    if(wv_seq[0] == 0 or wv_seq[0] == 3):
      if(a9_wv_weldingon==True):
        program_weld_on = False
        if(isHicomm):
          write_port_register(202,0)
          write_port_register(149,0)
        else:
          set_standard_digital_out(0,False)
        end
        if(wv_weldpar[2]==1):
          target_pos = feature_offset(get_actual_tcp_pose(),p[0,0,-0.01,0,0,0],wv_Line_Feature2)
          movel(target_pos,0.5,0.01)
        end
      end
    end
    background_pose = [dumy_p,dumy_p,dumy_p]
    move_p = background_pose
    return sin_dir
  end
  $ 147 "Reset"
  $ 148 "If Reset_Trig"
  if (Reset_Trig):
    $ 149 "Reset_Trig≔ False "
    global Reset_Trig=  False
    $ 150 "Call robotand_cell_initalizat"
    robotand_cell_initalizat()
    $ 151 "Auto_trig≔ False "
    global Auto_trig=  False
    $ 152 "write_port_register(cell_3f_2f_151,0)"
    write_port_register(cell_3f_2f_151,0)
    $ 153 "write_port_register(cell_info_152,0)"
    write_port_register(cell_info_152,0)
    $ 154 "write_port_register(weld_req_153,0)"
    write_port_register(weld_req_153,0)
    $ 155 "write_port_register(return_done_240,0)"
    write_port_register(return_done_240,0)
    $ 156 "write_port_register(robot_move_163,0)"
    write_port_register(robot_move_163,0)
    $ 157 "write_port_register(robot_pose_164,0)"
    write_port_register(robot_pose_164,0)
    $ 158 "write_port_register(182,0)"
    write_port_register(182,0)
    $ 159 "write_port_register(185,0)"
    write_port_register(185,0)
    $ 160 "write_port_register(201,0)"
    write_port_register(201,0)
    $ 161 "write_port_register(202,0)"
    write_port_register(202,0)
  end
  $ 162 "Welding_Init"
  $ 163 "'welding parameter initialization'"
  # 'welding parameter initialization'
  $ 164 "welding_etc"
  $ 192 "c5_wv_gap_y≔0"
  global c5_wv_gap_y=0
  $ 193 "c6_wv_gap_cpm≔0"
  global c6_wv_gap_cpm=0
  $ 194 "c9_wv_gap_freq≔0"
  global c9_wv_gap_freq=0
  $ 195 "c4_gap_enable≔0"
  global c4_gap_enable=0
  $ 196 "c7_wv_gap≔[c4_gap_enable,c5_wv_gap_y,c6_wv_gap_cpm,c9_wv_gap_freq]"
  global c7_wv_gap=[c4_gap_enable,c5_wv_gap_y,c6_wv_gap_cpm,c9_wv_gap_freq]
  $ 197 "init_reset_modbus_server"
  $ 198 "set_tool_voltage(24)"
  set_tool_voltage(24)
  $ 199 "write_port_register(163,0)"
  write_port_register(163,0)
  $ 200 "write_port_register(164,0)"
  write_port_register(164,0)
  $ 202 "write_port_register(201,1)"
  write_port_register(201,1)
  $ 203 "write_port_register(202,0)"
  write_port_register(202,0)
  $ 1257 "Thread_2"
  thread Thread_2():
    while (True):
      $ 1258 "heartbeat≔heartbeat+1"
      global heartbeat=heartbeat+1
      $ 1259 "If heartbeat>499"
      if (heartbeat>499):
        $ 1260 "heartbeat≔0"
        global heartbeat=0
      end
      $ 1261 "write_port_register(128,heartbeat)"
      write_port_register(128,heartbeat)
      $ 1271 "Wait: 1.0"
      sleep(1.0)
    end
  end
  threadId_Thread_2 = run Thread_2()
  $ 1272 "Thread_1"
  thread Thread_1():
    while (True):
      $ 1273 "a0_Job_Mode≔read_port_register(162)"
      global a0_Job_Mode= read_port_register (162)
      $ 1274 "a1_job_move≔read_port_register(163)"
      global a1_job_move= read_port_register (163)
      $ 1275 "If red_led≟ True "
      if (get_tool_digital_out(0) ==   True  ):
        $ 1276 "Set red_led=Off"
        set_tool_digital_out(0, False)
      end
      $ 1277 "If a0_Job_Mode≟2"
      if (a0_Job_Mode == 2):
        $ 1278 "If read_port_register(arc_onoff_168)≟2"
        if ( read_port_register (arc_onoff_168) == 2):
          $ 1279 "a9_wv_weldingon≔ True "
          global a9_wv_weldingon=  True
        else:
          $ 1280 "Else" "noBreak"
          $ 1281 "a9_wv_weldingon≔ False "
          global a9_wv_weldingon=  False
        end
        $ 1282 "If Auto_trig"
        if (Auto_trig):
          $ 1283 "get_next_number≔read_port_register(166)"
          global get_next_number= read_port_register (166)
          $ 1284 "get_move_trig≔read_port_register(167)"
          global get_move_trig= read_port_register (167)
          $ 1285 "If get_move_trig≟1 and running_trig≟ True "
          if (get_move_trig == 1  and  running_trig ==   True  ):
            $ 1286 "If get_next_number<0 or get_next_number>30"
            if (get_next_number<0  or  get_next_number>30):
              $ 1287 "write_port_register(142,141)"
              write_port_register(142,141)
              $ 1288 "Halt"
              halt
            end
            $ 1289 "If get_next_number≠Auto_cur_cell"
            if (get_next_number != Auto_cur_cell):
              $ 1290 "running_trig≔ False "
              global running_trig=  False
              $ 1291 "write_welder(0, False )"
              write_welder(0,  False  )
              $ 1292 "write_port_register(149,0)"
              write_port_register(149,0)
              $ 1293 "write_port_register(202,0)"
              write_port_register(202,0)
            else:
              $ 1294 "Else" "noBreak"
              $ 1295 "write_port_register(166,0)"
              write_port_register(166,0)
              $ 1296 "write_port_register(167,0)"
              write_port_register(167,0)
            end
          end
        end
        $ 1297 "If t_time>timer_1"
        if (t_time>timer_1):
          $ 1298 "write_port_register(143,timer_1)"
          write_port_register(143,timer_1)
        else:
          $ 1299 "Else" "noBreak"
          $ 1300 "write_port_register(143,timer_1)"
          write_port_register(143,timer_1)
          $ 1301 "write_port_register(144,timer_1)"
          write_port_register(144,timer_1)
        end
        $ 1302 "Monitoring touch and welding"
        $ 1303 "If read_welder_control(0) and read_port_register(130)≠1"
        if (read_welder_control(0)  and   read_port_register (130) != 1):
          $ 1304 "write_port_register(130,1)"
          write_port_register(130,1)
        else:
          $ 1305 "ElseIf read_welder_control(0) and read_port_register(130)≠0"
          if (read_welder_control(0)  and   read_port_register (130) != 0):
            $ 1306 "write_port_register(130,0)"
            write_port_register(130,0)
          end
        end
        $ 1307 "If read_welder(5)"
        if (read_welder(5)):
          $ 1308 "'check wcr in (digital)'"
          # 'check wcr in (digital)'
          $ 1309 "write_output_float_register(20,1)"
          write_output_float_register(20,1)
        else:
          $ 1310 "Else" "noBreak"
          $ 1311 "write_output_float_register(20,0)"
          write_output_float_register(20,0)
        end
        $ 1312 "If read_welder(4)"
        if (read_welder(4)):
          $ 1313 "'check touch (digital)'"
          # 'check touch (digital)'
          $ 1314 "write_output_float_register(21,1)"
          write_output_float_register(21,1)
        else:
          $ 1315 "Else" "noBreak"
          $ 1316 "write_output_float_register(21,0)"
          write_output_float_register(21,0)
        end
        $ 1317 "If read_welder_control(0)"
        if (read_welder_control(0)):
          $ 1318 "'check welding out (digital)'"
          # 'check welding out (digital)'
          $ 1319 "write_output_float_register(17,1)"
          write_output_float_register(17,1)
        else:
          $ 1320 "Else" "noBreak"
          $ 1321 "write_output_float_register(17,0)"
          write_output_float_register(17,0)
        end
        $ 1322 "If read_welder_control(4)"
        if (read_welder_control(4)):
          $ 1323 "'check touch out (digital)'"
          # 'check touch out (digital)'
          $ 1324 "write_output_float_register(18,1)"
          write_output_float_register(18,1)
        else:
          $ 1325 "Else" "noBreak"
          $ 1326 "write_output_float_register(18,0)"
          write_output_float_register(18,0)
        end
      end
      $ 1327 "If get_tool_digital_in(1)≟ True "
      if (get_tool_digital_in(1) ==   True  ):
        $ 1328 "set_tool_digital_out(1, False )"
        set_tool_digital_out(1,  False  )
      else:
        $ 1329 "Else" "noBreak"
        $ 1330 "set_tool_digital_out(1, True )"
        set_tool_digital_out(1,  True  )
      end
      $ 1331 "If red_led≟ True "
      if (get_tool_digital_out(0) ==   True  ):
        $ 1332 "Set red_led=Off"
        set_tool_digital_out(0, False)
        $ 1333 "end_freedrive_mode()"
        end_freedrive_mode()
      end
      $ 1334 "check_speed()"
      check_speed()
      $ 1335 "Wait: 0.05"
      sleep(0.05)
    end
  end
  threadId_Thread_1 = run Thread_1()
  thread EventThread():
    while (True):
      if (event_cal_on):
        $ 1339 "move_i_f≔1"
        global move_i_f=1
        $ 1340 "get_pose_side≔0"
        global get_pose_side=0
        $ 1341 "Loop move_i_f<10"
        while (move_i_f<10):
          $ 1342 "If A_Touch_trig_l[move_i_f]≟ True "
          if (A_Touch_trig_l[move_i_f] ==   True  ):
            $ 1343 "If move_i_f≟A_VL1 or move_i_f≟A_VL2"
            if (move_i_f == A_VL1  or  move_i_f == A_VL2):
              $ 1344 "A_sel_v≔move_i_f"
              global A_sel_v=move_i_f
              $ 1345 "If simulation_mode"
              if (simulation_mode):
                $ 1346 "Call welding_parameter_sim"
                welding_parameter_sim()
              else:
                $ 1347 "Else" "noBreak"
                $ 1348 "Call welding_parameter_init"
                welding_parameter_init()
              end
              $ 1349 "If a8_wv_distance<5"
              if (a8_wv_distance<5):
                $ 1350 "write_port_register(142,143)"
                write_port_register(142,143)
                $ 1351 "Halt"
                halt
              end
              $ 1352 "b2_left_par≔ True "
              global b2_left_par=  True
              $ 1353 "b8_wv_2f≔ False "
              global b8_wv_2f=  False
              $ 1354 "If move_i_f≟A_VL2"
              if (move_i_f == A_VL2):
                $ 1355 "callar_hor≔a6_callar_hor"
                global callar_hor=a6_callar_hor
                $ 1356 "b2_cell≔0"
                global b2_cell=0
                $ 1357 "If b1_cell_info_L≟c or b1_cell_info_L≟d or b1_cell_info_L≟E or b1_cell_info_L≟e"
                if (b1_cell_info_L == c  or  b1_cell_info_L == d  or  b1_cell_info_L == E  or  b1_cell_info_L == e):
                  $ 1358 "b2_cell≔b1_cell_info_L"
                  global b2_cell=b1_cell_info_L
                else:
                  $ 1359 "Else" "noBreak"
                  $ 1360 "b2_cell≔0"
                  global b2_cell=0
                end
              else:
                $ 1361 "Else" "noBreak"
                $ 1362 "callar_hor≔0"
                global callar_hor=0
                $ 1363 "b2_cell≔b1_cell_info_L"
                global b2_cell=b1_cell_info_L
              end
              $ 1364 "get_pos≔get_lr(left,a6_f_width,a5_f_hole,a7_f_distance,b2_left_par,b8_wv_2f,Touch_dis,get_margin_z,get_pose_side,callar_hor,b2_cell,center_line)"
              global get_pos=get_lr(p[.480496318984, .411279115151, .006998291210, -2.211681476386, -.899147924387, -1.383032568605],a6_f_width,a5_f_hole,a7_f_distance,b2_left_par,b8_wv_2f,Touch_dis,get_margin_z,get_pose_side,callar_hor,b2_cell,center_line)
              $ 1365 "pre_tp≔tilt_3f_fun(get_pos,[0,0,0],0)"
              global pre_tp=tilt_3f_fun(get_pos,[0,0,0],0)
              $ 1366 "A_Prepos_l[move_i_f]=pre_tp"
              A_Prepos_l[move_i_f]=pre_tp
            else:
              $ 1367 "ElseIf move_i_f≟A_VR1 or move_i_f≟A_VR2"
              if (move_i_f == A_VR1  or  move_i_f == A_VR2):
                $ 1368 "A_sel_v≔move_i_f"
                global A_sel_v=move_i_f
                $ 1369 "If simulation_mode"
                if (simulation_mode):
                  $ 1370 "Call welding_parameter_sim"
                  welding_parameter_sim()
                else:
                  $ 1371 "Else" "noBreak"
                  $ 1372 "Call welding_parameter_init"
                  welding_parameter_init()
                end
                $ 1373 "If a8_wv_distance<5"
                if (a8_wv_distance<5):
                  $ 1374 "write_port_register(142,143)"
                  write_port_register(142,143)
                  $ 1375 "Halt"
                  halt
                end
                $ 1376 "b2_left_par≔ False "
                global b2_left_par=  False
                $ 1377 "b8_wv_2f≔ False "
                global b8_wv_2f=  False
                $ 1378 "If move_i_f≟A_VR2"
                if (move_i_f == A_VR2):
                  $ 1379 "callar_hor≔a6_callar_hor"
                  global callar_hor=a6_callar_hor
                  $ 1380 "If b1_cell_info_R≟c or b1_cell_info_R≟d or b1_cell_info_R≟E or b1_cell_info_R≟e"
                  if (b1_cell_info_R == c  or  b1_cell_info_R == d  or  b1_cell_info_R == E  or  b1_cell_info_R == e):
                    $ 1381 "b2_cell≔b1_cell_info_R"
                    global b2_cell=b1_cell_info_R
                  else:
                    $ 1382 "Else" "noBreak"
                    $ 1383 "b2_cell≔0"
                    global b2_cell=0
                  end
                else:
                  $ 1384 "Else" "noBreak"
                  $ 1385 "callar_hor≔0"
                  global callar_hor=0
                  $ 1386 "b2_cell≔b1_cell_info_R"
                  global b2_cell=b1_cell_info_R
                end
                $ 1387 "get_pos≔get_lr(right,a6_f_width,a5_f_hole,a7_f_distance,b2_left_par,b8_wv_2f,Touch_dis,get_margin_z,get_pose_side,callar_hor,b2_cell,center_line)"
                global get_pos=get_lr(p[.475000000000, -.421403215678, .026417194146, 1.917761036827, -1.141682393512, 1.523356199292],a6_f_width,a5_f_hole,a7_f_distance,b2_left_par,b8_wv_2f,Touch_dis,get_margin_z,get_pose_side,callar_hor,b2_cell,center_line)
                $ 1388 "pre_tp≔tilt_3f_fun(get_pos,[0,0,0],0)"
                global pre_tp=tilt_3f_fun(get_pos,[0,0,0],0)
                $ 1389 "A_Prepos_l[move_i_f]=pre_tp"
                A_Prepos_l[move_i_f]=pre_tp
              else:
                $ 1390 "ElseIf move_i_f≟A_HOR"
                if (move_i_f == A_HOR):
                  $ 1391 "A_sel_v≔A_HOR"
                  global A_sel_v=A_HOR
                  $ 1392 "If simulation_mode"
                  if (simulation_mode):
                    $ 1393 "Call welding_parameter_sim"
                    welding_parameter_sim()
                  else:
                    $ 1394 "Else" "noBreak"
                    $ 1395 "Call welding_parameter_init"
                    welding_parameter_init()
                  end
                  $ 1396 "b8_wv_2f≔ True "
                  global b8_wv_2f=  True
                  $ 1397 "b2_left_par≔ True "
                  global b2_left_par=  True
                  $ 1398 "b2_cell≔b1_cell_info_L"
                  global b2_cell=b1_cell_info_L
                  $ 1399 "get_pos≔get_lr(up_left,a6_f_width,a5_f_hole,a7_f_distance,b2_left_par,b8_wv_2f,Touch_dis,get_margin_z,get_pose_side,0,b2_cell,center_line)"
                  global get_pos=get_lr(p[.492775857339, .409517380626, -.029063830209, -2.419264859926, -.998084331190, -1.368689080860],a6_f_width,a5_f_hole,a7_f_distance,b2_left_par,b8_wv_2f,Touch_dis,get_margin_z,get_pose_side,0,b2_cell,center_line)
                  $ 1400 "pre_tp≔get_pos"
                  global pre_tp=get_pos
                  $ 1401 "A_Prepos_l[move_i_f]=pre_tp"
                  A_Prepos_l[move_i_f]=pre_tp
                else:
                  $ 1402 "ElseIf move_i_f≟A_HOR_R"
                  if (move_i_f == A_HOR_R):
                    $ 1403 "A_sel_v≔A_HOR"
                    global A_sel_v=A_HOR
                    $ 1404 "If simulation_mode"
                    if (simulation_mode):
                      $ 1405 "Call welding_parameter_sim"
                      welding_parameter_sim()
                    else:
                      $ 1406 "Else" "noBreak"
                      $ 1407 "Call welding_parameter_init"
                      welding_parameter_init()
                    end
                    $ 1408 "b2_left_par≔ False "
                    global b2_left_par=  False
                    $ 1409 "b8_wv_2f≔ True "
                    global b8_wv_2f=  True
                    $ 1410 "b2_cell≔b1_cell_info_R"
                    global b2_cell=b1_cell_info_R
                    $ 1411 "get_pos≔get_lr(up_right,a6_f_width,a5_f_hole,a7_f_distance,b2_left_par,b8_wv_2f,Touch_dis,get_margin_z,get_pose_side,0,b2_cell,center_line)"
                    global get_pos=get_lr(p[.445203173045, -.406687378356, -.031125942276, 2.308490741423, -1.066468937023, 1.322151316133],a6_f_width,a5_f_hole,a7_f_distance,b2_left_par,b8_wv_2f,Touch_dis,get_margin_z,get_pose_side,0,b2_cell,center_line)
                    $ 1412 "pre_tp≔get_pos"
                    global pre_tp=get_pos
                    $ 1413 "A_Prepos_l[move_i_f]=pre_tp"
                    A_Prepos_l[move_i_f]=pre_tp
                  else:
                    $ 1414 "ElseIf move_i_f≟A_HOR_ML"
                    if (move_i_f == A_HOR_ML):
                      $ 1415 "A_sel_v≔A_HOR_ML"
                      global A_sel_v=A_HOR_ML
                      $ 1416 "If simulation_mode"
                      if (simulation_mode):
                        $ 1417 "Call welding_parameter_sim"
                        welding_parameter_sim()
                      else:
                        $ 1418 "Else" "noBreak"
                        $ 1419 "Call welding_parameter_init"
                        welding_parameter_init()
                      end
                      $ 1420 "b8_wv_2f≔ True "
                      global b8_wv_2f=  True
                      $ 1421 "b2_left_par≔ True "
                      global b2_left_par=  True
                      $ 1422 "b2_cell≔b1_cell_info_L"
                      global b2_cell=b1_cell_info_L
                      $ 1423 "Touch_dis≔-1*Touch_dis"
                      global Touch_dis=-1*Touch_dis
                      $ 1424 "get_pos≔get_lr(up_left,a6_f_width,a5_f_hole,a7_f_distance,b2_left_par,b8_wv_2f,Touch_dis,get_margin_z,get_pose_side,a6_callar_hor,b2_cell,center_line)"
                      global get_pos=get_lr(p[.492775857339, .409517380626, -.029063830209, -2.419264859926, -.998084331190, -1.368689080860],a6_f_width,a5_f_hole,a7_f_distance,b2_left_par,b8_wv_2f,Touch_dis,get_margin_z,get_pose_side,a6_callar_hor,b2_cell,center_line)
                      $ 1425 "Touch_dis≔-1*Touch_dis"
                      global Touch_dis=-1*Touch_dis
                      $ 1426 "pre_tp≔get_pos"
                      global pre_tp=get_pos
                      $ 1427 "A_Prepos_l[move_i_f]=pre_tp"
                      A_Prepos_l[move_i_f]=pre_tp
                    else:
                      $ 1428 "ElseIf move_i_f≟A_HOR_MR"
                      if (move_i_f == A_HOR_MR):
                        $ 1429 "A_sel_v≔A_HOR_MR"
                        global A_sel_v=A_HOR_MR
                        $ 1430 "If simulation_mode"
                        if (simulation_mode):
                          $ 1431 "Call welding_parameter_sim"
                          welding_parameter_sim()
                        else:
                          $ 1432 "Else" "noBreak"
                          $ 1433 "Call welding_parameter_init"
                          welding_parameter_init()
                        end
                        $ 1434 "b2_left_par≔ False "
                        global b2_left_par=  False
                        $ 1435 "b8_wv_2f≔ True "
                        global b8_wv_2f=  True
                        $ 1436 "b2_cell≔b1_cell_info_R"
                        global b2_cell=b1_cell_info_R
                        $ 1437 "Touch_dis≔-1*Touch_dis"
                        global Touch_dis=-1*Touch_dis
                        $ 1438 "get_pos≔get_lr(up_right,a6_f_width,a5_f_hole,a7_f_distance,b2_left_par,b8_wv_2f,Touch_dis,get_margin_z,get_pose_side,a6_callar_hor,b2_cell,center_line)"
                        global get_pos=get_lr(p[.445203173045, -.406687378356, -.031125942276, 2.308490741423, -1.066468937023, 1.322151316133],a6_f_width,a5_f_hole,a7_f_distance,b2_left_par,b8_wv_2f,Touch_dis,get_margin_z,get_pose_side,a6_callar_hor,b2_cell,center_line)
                        $ 1439 "Touch_dis≔-1*Touch_dis"
                        global Touch_dis=-1*Touch_dis
                        $ 1440 "pre_tp≔get_pos"
                        global pre_tp=get_pos
                        $ 1441 "A_Prepos_l[move_i_f]=pre_tp"
                        A_Prepos_l[move_i_f]=pre_tp
                      end
                    end
                  end
                end
              end
            end
            $ 1442 "If move_i_f≤4"
            if (move_i_f <= 4):
              $ 1443 "A_Prepos_l[move_i_f+9]=p[0,0,0,0,0,0]"
              A_Prepos_l[move_i_f+9]=p[0,0,0,0,0,0]
            end
          end
          $ 1446 "move_i_f≔move_i_f+1"
          global move_i_f=move_i_f+1
        end
        $ 1447 "event_cal_on≔ False "
        global event_cal_on=  False
      elif (event_side_on):
        $ 1451 "Wait event_cal_on≟ False "
        while (not(event_cal_on ==   False  )):
          sync()
        end
        $ 1452 "move_i_f≔1"
        global move_i_f=1
        $ 1453 "get_pose_side≔get_pose_side_t"
        global get_pose_side=get_pose_side_t
        $ 1454 "Loop move_i_f<10"
        while (move_i_f<10):
          $ 1455 "If A_Touch_trig_l[move_i_f]≟ True "
          if (A_Touch_trig_l[move_i_f] ==   True  ):
            $ 1456 "If move_i_f≟A_VL1 or move_i_f≟A_VL2"
            if (move_i_f == A_VL1  or  move_i_f == A_VL2):
              $ 1457 "A_Prepos_l[move_i_f]=side_apply(A_Prepos_l[move_i_f],center_line,get_pose_side)"
              A_Prepos_l[move_i_f]=side_apply(A_Prepos_l[move_i_f],center_line,get_pose_side)
            else:
              $ 1458 "ElseIf move_i_f≟A_VR1 or move_i_f≟A_VR2"
              if (move_i_f == A_VR1  or  move_i_f == A_VR2):
                $ 1459 "A_Prepos_l[move_i_f]=side_apply(A_Prepos_l[move_i_f],center_line,get_pose_side)"
                A_Prepos_l[move_i_f]=side_apply(A_Prepos_l[move_i_f],center_line,get_pose_side)
              else:
                $ 1460 "ElseIf move_i_f≟A_HOR"
                if (move_i_f == A_HOR):
                  $ 1461 "A_Prepos_l[move_i_f]=side_apply(A_Prepos_l[move_i_f],center_line,get_pose_side)"
                  A_Prepos_l[move_i_f]=side_apply(A_Prepos_l[move_i_f],center_line,get_pose_side)
                else:
                  $ 1462 "ElseIf move_i_f≟A_HOR_R"
                  if (move_i_f == A_HOR_R):
                    $ 1463 "A_Prepos_l[move_i_f]=side_apply(A_Prepos_l[move_i_f],center_line,get_pose_side)"
                    A_Prepos_l[move_i_f]=side_apply(A_Prepos_l[move_i_f],center_line,get_pose_side)
                  else:
                    $ 1464 "ElseIf move_i_f≟A_HOR_ML"
                    if (move_i_f == A_HOR_ML):
                      $ 1465 "A_Prepos_l[move_i_f]=side_apply(A_Prepos_l[move_i_f],center_line,get_pose_side)"
                      A_Prepos_l[move_i_f]=side_apply(A_Prepos_l[move_i_f],center_line,get_pose_side)
                    else:
                      $ 1466 "ElseIf move_i_f≟A_HOR_MR"
                      if (move_i_f == A_HOR_MR):
                        $ 1467 "A_Prepos_l[move_i_f]=side_apply(A_Prepos_l[move_i_f],center_line,get_pose_side)"
                        A_Prepos_l[move_i_f]=side_apply(A_Prepos_l[move_i_f],center_line,get_pose_side)
                      end
                    end
                  end
                end
              end
            end
          end
          $ 1468 "move_i_f≔move_i_f+1"
          global move_i_f=move_i_f+1
        end
        $ 1469 "event_side_on≔ False "
        global event_side_on=  False
      elif (reset_trig):
        $ 1471 "Call reset_weld_param"
        reset_weld_param()
        $ 1472 "reset_trig≔ False "
        global reset_trig=  False
      elif (time_cal_trig):
        $ 1474 "t_time≔time_cal(Auto_W_num,Auto_total_cell,A_Speed_list,A_Distance_list,A_Touch_p,0)"
        global t_time=time_cal(Auto_W_num,Auto_total_cell,A_Speed_list,A_Distance_list,A_Touch_p,0)
        $ 1475 "write_port_register(144,t_time)"
        write_port_register(144,t_time)
        $ 1476 "time_cal_trig≔ False "
        global time_cal_trig=  False
      elif (pause_trig):
        $ 1478 "s_conn≔socket_open('192.168.1.7',29999)"
        global s_conn=socket_open("192.168.1.7",29999)
        $ 1479 "s_send≔socket_send_string('pause')"
        global s_send=socket_send_string("pause")
        $ 1480 "s_send≔socket_send_byte(10)"
        global s_send=socket_send_byte(10)
        $ 1481 "socket_close()"
        socket_close()
        $ 1482 "pause_trig≔ False "
        global pause_trig=  False
      end
      sync()
    end
  end
  eventThread = run EventThread()
  while (True):
    $ 204 "Robot Program"
    $ 222 "If simulation_mode"
    if (simulation_mode):
      $ 223 "'work mode 2'"
      # 'work mode 2'
      $ 224 "write_port_register(162,2)"
      write_port_register(162,2)
      $ 225 "touch_temp≔0"
      global touch_temp=0
    end
    $ 226 "If a0_Job_Mode≟1"
    if (a0_Job_Mode == 1):
      $ 227 "job mode 1"
      $ 228 "'JOB_MANUAL'"
      # 'JOB_MANUAL'
      $ 229 "write_port_register(robot_ready_141,1)"
      write_port_register(robot_ready_141,1)
      $ 230 "If freedrive≟ True  and freedrive_trg≟ False "
      if (get_tool_digital_in(1) ==   True    and  freedrive_trg ==   False  ):
        $ 231 "freedrive_trg≔ True "
        global freedrive_trg=  True
        $ 232 "freedrive_mode()"
        freedrive_mode()
      else:
        $ 233 "ElseIf freedrive≟ False  and freedrive_trg≟ True "
        if (get_tool_digital_in(1) ==   False    and  freedrive_trg ==   True  ):
          $ 234 "end_freedrive_mode()"
          end_freedrive_mode()
          $ 235 "freedrive_trg≔ False "
          global freedrive_trg=  False
        end
      end
      $ 239 "If freedrive≟ True  and save_tool≟ True "
      if (get_tool_digital_in(1) ==   True    and  get_tool_digital_in(0) ==   True  ):
        $ 243 "Wait: 0.01"
        sleep(0.01)
      else:
        $ 244 "ElseIf a1_job_move≟1"
        if (a1_job_move == 1):
          $ 245 "'Manual - Move Home/Packing/Warmup'"
          # 'Manual - Move Home/Packing/Warmup'
          $ 246 "If read_port_register(robot_pose_164)≟1"
          if ( read_port_register (robot_pose_164) == 1):
            $ 247 "write_port_register(robot_ready_141,0)"
            write_port_register(robot_ready_141,0)
            $ 248 "homeing()"
            homeing()
            $ 249 "MoveJ"
            $ 250 "Packing_pos" "breakAfter"
            movej([1.5877798795700073, -0.0173419157611292, -2.4983108679400843, -1.4065726439105433, 1.626846194267273, 3.0169763565063477], a=0.9599310885968813, v=0.9599310885968813)
          else:
            $ 251 "ElseIf read_port_register(robot_pose_164)≟2"
            if ( read_port_register (robot_pose_164) == 2):
              $ 252 "write_port_register(robot_ready_141,0)"
              write_port_register(robot_ready_141,0)
              $ 253 "homeing()"
              homeing()
            else:
              $ 254 "ElseIf read_port_register(robot_pose_164)≟3"
              global thread_flag_254=0
              thread Thread_if_254():
                $ 255 "write_port_register(robot_ready_141,0)"
                write_port_register(robot_ready_141,0)
                $ 256 "Warm-up"
                $ 257 "Loop 22 times"
                Loop_9 = 0
                while (Loop_9 < 22):
                  $ 258 "MoveJ"
                  $ 259 "Warming_1" "breakAfter"
                  movej([1.3388409470167426, -1.0894445773085817, -1.21578769245379, -2.340308120379028, 1.4975742894997062, 2.3546781160711117], a=0.5235987755982988, v=0.2617993877991494)
                  $ 260 "Warming_2" "breakAfter"
                  movej([0.3765170846483107, -1.0894466320678031, -1.215768207322279, -2.3402268007341895, 1.4977834941028334, 2.3545507363355367], a=0.5235987755982988, v=0.2617993877991494)
                  $ 261 "Warming_3" "breakAfter"
                  movej([0.70229908534082, -1.0894474234917375, -1.2158576930717002, -2.340314378048955, 1.497725846219038, 2.3545705560997385], a=0.5235987755982988, v=0.2617993877991494)
                  $ 262 "Warming_4" "breakAfter"
                  movej([0.7262700130956564, -1.3120291852612347, -1.2099656497338014, -2.3525900953229293, 1.4887798341942113, 2.3787312683819053], a=0.5235987755982988, v=0.2617993877991494)
                  $ 263 "Wariming_5" "breakAfter"
                  movej([0.6926726182060315, -1.0476106481659855, -1.2179788018883642, -2.3355421428203886, 1.501172277634622, 2.3452576869092923], a=0.5235987755982988, v=0.2617993877991494)
                  $ 264 "Warming_6" "breakAfter"
                  movej([0.706544616734295, -1.047040496424307, -1.4190888321133315, -2.3436933501169452, 1.4896422361111494, 2.359727124413684], a=0.5235987755982988, v=0.2617993877991494)
                  $ 265 "Warming_7" "breakAfter"
                  movej([0.6929880468286825, -1.0476354157293724, -1.2203987593812862, -2.335678707355349, 1.5010671072282735, 2.34550338764565], a=0.5235987755982988, v=0.2617993877991494)
                  $ 266 "Warming_8" "breakAfter"
                  movej([0.6920775233962951, -1.0506328608604214, -1.2152130579572011, -2.5072867131215766, 1.4917910996963177, 2.3459413556024855], a=0.5235987755982988, v=0.2617993877991494)
                  $ 267 "Warming_9" "breakAfter"
                  movej([0.692933302781529, -1.0474869681006531, -1.2206503884398048, -2.327559666709858, 1.5015191668476027, 2.3454614641680087], a=0.5235987755982988, v=0.2617993877991494)
                  $ 268 "Warming_10" "breakAfter"
                  movej([0.7189566793816887, -1.1462083943843844, -1.3286482352122917, -2.3898368690561114, 1.223390234561962, 2.3705741030878644], a=0.5235987755982988, v=0.2617993877991494)
                  $ 269 "Warming_11" "breakAfter"
                  movej([0.6952417412291937, -1.0226626805382075, -1.3187663864026051, -2.3852732107244847, 1.5281305955128988, 2.3484138521676003], a=0.5235987755982988, v=0.2617993877991494)
                  $ 270 "Warming_12" "breakAfter"
                  movej([0.6939658935868351, -1.0222541193887693, -1.3205060700309819, -2.4036431483224994, 1.8876292979334401, 2.3447872177861786], a=0.5235987755982988, v=0.2617993877991494)
                  $ 271 "Warming_13" "breakAfter"
                  movej([0.6855475262233561, -1.0389108716421376, -1.3163550590643318, -2.371185255756596, 1.5282046997566647, 1.6427118007650936], a=0.5235987755982988, v=0.2617993877991494)
                  $ 272 "Warming_14" "breakAfter"
                  movej([0.721349856763205, -1.0075982028648234, -1.3205933019427434, -2.399656340024448, 1.5281938267886401, 2.9170078642332813], a=0.5235987755982988, v=0.2617993877991494)
                  Loop_9 = Loop_9 + 1
                end
                $ 273 "homeing()"
                homeing()
                $ 274 "Wait: 2.0"
                sleep(2.0)
                thread_flag_254 = 1
              end
              if ( read_port_register (robot_pose_164) == 3):
                global thread_handler_254=run Thread_if_254()
                while (thread_flag_254 == 0):
                  if not( read_port_register (robot_pose_164) == 3):
                    kill thread_handler_254
                    thread_flag_254 = 2
                  else:
                    sync()
                  end
                end
              else:
                thread_flag_254 = 2
              end
              if (thread_flag_254 == 2):
                $ 275 "ElseIf read_port_register(robot_pose_164)≟4"
                if ( read_port_register (robot_pose_164) == 4):
                  $ 276 "write_port_register(robot_ready_141,0)"
                  write_port_register(robot_ready_141,0)
                  $ 277 "homeing()"
                  homeing()
                  $ 278 "MoveJ"
                  $ 279 "pre_mounting" "breakAfter"
                  movej([1.2356762886047363, -0.8703244368182581, -0.942230526600973, -2.3905327955829065, 1.3216267824172974, 2.6514604091644287], a=0.7853981633974483, v=0.7853981633974483)
                  $ 280 "Mounting_pos" "breakAfter"
                  movej([0.6231353085164267, -0.6300961531972575, -0.9034285948871803, -1.770059340221131, 1.417516049558281, 1.7792033261567348], a=0.7853981633974483, v=0.7853981633974483)
                else:
                  $ 281 "ElseIf read_port_register(robot_pose_164)≟5"
                  if ( read_port_register (robot_pose_164) == 5):
                    $ 282 "c_p≔get_actual_tcp_pose()"
                    global c_p= get_actual_tcp_pose ()
                    $ 283 "MoveL"
                    $ 284 "m_p≔pose_trans(c_p, p[0,0,0,d2r(tilt_deg_man),0,0])"
                    global m_p= pose_trans (c_p, p[0,0,0,d2r(tilt_deg_man),0,0])
                    $ 285 "m_p" "breakAfter"
                    movel(pose_trans(Base, m_p), a=0.03, v=0.03)
                    $ 286 "m_p≔pose_trans(c_p, p[0,0,0,d2r(-tilt_deg_man),0,0])"
                    global m_p= pose_trans (c_p, p[0,0,0,d2r(-tilt_deg_man),0,0])
                    $ 287 "m_p" "breakAfter"
                    movel(pose_trans(Base, m_p), a=0.03, v=0.03)
                    $ 288 "c_p" "breakAfter"
                    movel(pose_trans(Base, c_p), a=0.03, v=0.03)
                    $ 289 "m_p≔pose_trans(c_p, p[0,0,0,0,d2r(tilt_deg_man),0])"
                    global m_p= pose_trans (c_p, p[0,0,0,0,d2r(tilt_deg_man),0])
                    $ 290 "m_p" "breakAfter"
                    movel(pose_trans(Base, m_p), a=0.03, v=0.03)
                    $ 291 "m_p≔pose_trans(c_p, p[0,0,0,0,d2r(-tilt_deg_man),0])"
                    global m_p= pose_trans (c_p, p[0,0,0,0,d2r(-tilt_deg_man),0])
                    $ 292 "m_p" "breakAfter"
                    movel(pose_trans(Base, m_p), a=0.03, v=0.03)
                    $ 293 "c_p" "breakAfter"
                    movel(pose_trans(Base, c_p), a=0.03, v=0.03)
                    $ 294 "m_p≔pose_trans(c_p, p[0,0,0,0,0,d2r(tilt_deg_man)])"
                    global m_p= pose_trans (c_p, p[0,0,0,0,0,d2r(tilt_deg_man)])
                    $ 295 "m_p" "breakAfter"
                    movel(pose_trans(Base, m_p), a=0.03, v=0.03)
                    $ 296 "m_p≔pose_trans(c_p, p[0,0,0,0,0,d2r(-tilt_deg_man)])"
                    global m_p= pose_trans (c_p, p[0,0,0,0,0,d2r(-tilt_deg_man)])
                    $ 297 "m_p" "breakAfter"
                    movel(pose_trans(Base, m_p), a=0.03, v=0.03)
                    $ 298 "c_p" "breakAfter"
                    movel(pose_trans(Base, c_p), a=0.03, v=0.03)
                  end
                end
              end
            end
          end
          $ 299 "Call Move_done"
          Move_done()
        end
      end
      $ 300 "Call robotand_cell_initalizat"
      robotand_cell_initalizat()
    else:
      $ 301 "ElseIf a0_Job_Mode≟2"
      global thread_flag_301=0
      thread Thread_if_301():
        $ 302 "'JOB_AUTO'"
        # 'JOB_AUTO'
        $ 303 "auto_on≔ True "
        global auto_on=  True
        $ 304 "Init"
        $ 305 "If freedrive_trg"
        if (freedrive_trg):
          $ 306 "end_freedrive_mode()"
          end_freedrive_mode()
          $ 307 "freedrive_trg≔ False "
          global freedrive_trg=  False
        end
        $ 308 "write_port_register(202,0)"
        write_port_register(202,0)
        $ 309 "write_port_register(robot_ready_141,0)"
        write_port_register(robot_ready_141,0)
        $ 310 "homeing()"
        homeing()
        $ 311 "Wait: 0.2"
        sleep(0.2)
        $ 312 "Cell_calculation"
        $ 313 "'setting'"
        # 'setting'
        $ 314 "Auto_trig≔ False "
        global Auto_trig=  False
        $ 315 "If Auto_trig≟ False "
        if (Auto_trig ==   False  ):
          $ 316 "If simulation_mode"
          if (simulation_mode):
            $ 317 "b1_cell_info_L≔B"
            global b1_cell_info_L=B
            $ 318 "b1_cell_info_R≔B"
            global b1_cell_info_R=B
            $ 319 "b1_cell_select≔motion_num([A_VL1,A_VR1,A_HOR,0,0,0])"
            global b1_cell_select=motion_num([A_VL1,A_VR1,A_HOR,0,0,0])
            $ 320 "b1_cell_select≔motion_num([A_HOR,0,0,0,0,0])"
            global b1_cell_select=motion_num([A_HOR,0,0,0,0,0])
            $ 321 "EXT_flag1≔integer_to_binary_list(read_port_register(2048))"
            global EXT_flag1= integer_to_binary_list ( read_port_register (2048))
            $ 322 "b1_cell_thickne≔6"
            global b1_cell_thickne=6
            $ 323 "A_Touch_trig_l≔touch_cal(b1_cell_info_L,b1_cell_info_R,b1_cell_select)"
            global A_Touch_trig_l=touch_cal(b1_cell_info_L,b1_cell_info_R,b1_cell_select)
            $ 324 "Auto_W_num≔cell_motion(A_Touch_trig_l,b1_cell_thickne,EXT_flag1,b1_cell_info_L,b1_cell_info_R)"
            global Auto_W_num=cell_motion(A_Touch_trig_l,b1_cell_thickne,EXT_flag1,b1_cell_info_L,b1_cell_info_R)
            $ 326 "Auto_total_cell≔cell_num(Auto_W_num)"
            global Auto_total_cell=cell_num(Auto_W_num)
            $ 327 "Auto_trig≔ True "
            global Auto_trig=  True
            $ 328 "A_sel_v≔Auto_W_num[0]"
            global A_sel_v=Auto_W_num[0]
          else:
            $ 329 "Else" "noBreak"
            $ 330 "b1_cell_info_L≔read_port_register(171)"
            global b1_cell_info_L= read_port_register (171)
            $ 331 "b1_cell_info_R≔read_port_register(172)"
            global b1_cell_info_R= read_port_register (172)
            $ 332 "EXT_flag1≔integer_to_binary_list(read_port_register(179))"
            global EXT_flag1= integer_to_binary_list ( read_port_register (179))
            $ 333 "b1_cell_select≔read_port_register(178)"
            global b1_cell_select= read_port_register (178)
            $ 334 "b1_cell_thickne≔read_port_register(183)"
            global b1_cell_thickne= read_port_register (183)
            $ 335 "A_Touch_trig_l≔touch_cal(b1_cell_info_L,b1_cell_info_R,b1_cell_select)"
            global A_Touch_trig_l=touch_cal(b1_cell_info_L,b1_cell_info_R,b1_cell_select)
            $ 336 "Auto_W_num≔cell_motion(A_Touch_trig_l,b1_cell_thickne,EXT_flag1,b1_cell_info_L,b1_cell_info_R)"
            global Auto_W_num=cell_motion(A_Touch_trig_l,b1_cell_thickne,EXT_flag1,b1_cell_info_L,b1_cell_info_R)
            $ 337 "Auto_total_cell≔cell_num(Auto_W_num)"
            global Auto_total_cell=cell_num(Auto_W_num)
            $ 338 "Auto_trig≔ True "
            global Auto_trig=  True
            $ 339 "A_sel_v≔Auto_W_num[0]"
            global A_sel_v=Auto_W_num[0]
          end
          $ 340 "write_port_register(139,Auto_total_cell-1)"
          write_port_register(139,Auto_total_cell-1)
        end
        $ 341 "Auto_cur_cell≔0"
        global Auto_cur_cell=0
        $ 342 "Touch,Welding"
        $ 343 "'Calculate total sequence and decide way'"
        # 'Calculate total sequence and decide way'
        $ 344 "Calculate & Move & Touch"
        $ 345 "touch_init"
        $ 346 "Call cell_info"
        cell_info()
        $ 347 "If simulation_mode"
        if (simulation_mode):
          $ 348 "Call welding_parameter_sim"
          welding_parameter_sim()
        else:
          $ 349 "Else" "noBreak"
          $ 350 "Call welding_parameter_init"
          welding_parameter_init()
          $ 351 "touch_temp≔read_port_register(180)"
          global touch_temp= read_port_register (180)
          $ 352 "A_cur_2f≔0"
          global A_cur_2f=0
          $ 353 "wv_direction≔1"
          global wv_direction=1
        end
        $ 354 "If touch_temp≟0"
        if (touch_temp == 0):
          $ 355 "reset Variable"
          $ 356 "A_Prepos_l=[p[0, 0, 0, 0, 0, 0], p[0, 0, 0, 0, 0, 0], p[0, 0, 0, 0, 0, 0],p[0, 0, 0, 0, 0, 0], p[0, 0, 0, 0, 0, 0], p[0, 0, 0, 0, 0, 0], p[0, 0, 0, 0, 0, 0], p[0, 0, 0, 0, 0, 0], p[0, 0, 0, 0, 0, 0], p[0, 0, 0, 0, 0, 0], p[0, 0, 0, 0, 0, 0],p[0, 0, 0, 0, 0, 0],p[0, 0, 0, 0, 0, 0],p[0, 0, 0, 0, 0, 0],p[0, 0, 0, 0, 0, 0],p[0,0,0,0,0,0]]"
          A_Prepos_l=[p[0, 0, 0, 0, 0, 0], p[0, 0, 0, 0, 0, 0], p[0, 0, 0, 0, 0, 0],p[0, 0, 0, 0, 0, 0], p[0, 0, 0, 0, 0, 0], p[0, 0, 0, 0, 0, 0], p[0, 0, 0, 0, 0, 0], p[0, 0, 0, 0, 0, 0], p[0, 0, 0, 0, 0, 0], p[0, 0, 0, 0, 0, 0], p[0, 0, 0, 0, 0, 0],p[0, 0, 0, 0, 0, 0],p[0, 0, 0, 0, 0, 0],p[0, 0, 0, 0, 0, 0],p[0, 0, 0, 0, 0, 0],p[0,0,0,0,0,0]]
          $ 357 "A_Touch_p=[p[0, 0, 0, 0, 0, 0], p[0, 0, 0, 0, 0, 0], p[0, 0, 0, 0, 0, 0],p[0, 0, 0, 0, 0, 0], p[0, 0, 0, 0, 0, 0], p[0, 0, 0, 0, 0, 0], p[0, 0, 0, 0, 0, 0], p[0, 0, 0, 0, 0, 0], p[0, 0, 0, 0, 0, 0], p[0, 0, 0, 0, 0, 0], p[0, 0, 0, 0, 0, 0],p[0, 0, 0, 0, 0, 0],p[0, 0, 0, 0, 0, 0],p[0, 0, 0, 0, 0, 0],p[0, 0, 0, 0, 0, 0],p[0,0,0,0,0,0]]"
          A_Touch_p=[p[0, 0, 0, 0, 0, 0], p[0, 0, 0, 0, 0, 0], p[0, 0, 0, 0, 0, 0],p[0, 0, 0, 0, 0, 0], p[0, 0, 0, 0, 0, 0], p[0, 0, 0, 0, 0, 0], p[0, 0, 0, 0, 0, 0], p[0, 0, 0, 0, 0, 0], p[0, 0, 0, 0, 0, 0], p[0, 0, 0, 0, 0, 0], p[0, 0, 0, 0, 0, 0],p[0, 0, 0, 0, 0, 0],p[0, 0, 0, 0, 0, 0],p[0, 0, 0, 0, 0, 0],p[0, 0, 0, 0, 0, 0],p[0,0,0,0,0,0]]
          $ 358 "reset_par"
          $ 359 "for_cal_rot≔p[0,0,0,0,0,0]"
          global for_cal_rot=p[0,0,0,0,0,0]
          $ 360 "for_cal_zr≔p[0,0,0,0,0,0]"
          global for_cal_zr=p[0,0,0,0,0,0]
          $ 361 "for_cal_zl≔p[0,0,0,0,0,0]"
          global for_cal_zl=p[0,0,0,0,0,0]
          $ 362 "for_cal_x_wel≔p[0,0,0,0,0,0]"
          global for_cal_x_wel=p[0,0,0,0,0,0]
          $ 363 "for_cal_xy≔p[0,0,0,0,0,0]"
          global for_cal_xy=p[0,0,0,0,0,0]
          $ 364 "for_cal_y_wel≔p[0,0,0,0,0,0]"
          global for_cal_y_wel=p[0,0,0,0,0,0]
          $ 365 "for_x_HOR≔p[0,0,0,0,0,0]"
          global for_x_HOR=p[0,0,0,0,0,0]
          $ 366 "for_x_HOR_R≔p[0,0,0,0,0,0]"
          global for_x_HOR_R=p[0,0,0,0,0,0]
          $ 367 "for_z_VL1≔p[0,0,0,0,0,0]"
          global for_z_VL1=p[0,0,0,0,0,0]
          $ 368 "for_z_VR1≔p[0,0,0,0,0,0]"
          global for_z_VR1=p[0,0,0,0,0,0]
        end
        $ 369 "write_port_register(143,0)"
        write_port_register(143,0)
        $ 370 "write_port_register(144,0)"
        write_port_register(144,0)
        $ 371 "timer_1: Reset"
        timer_1 = 0
        $ 372 "EXT_flag1≔integer_to_binary_list(read_port_register(179))"
        global EXT_flag1= integer_to_binary_list ( read_port_register (179))
        $ 374 "If touch_temp≟0"
        if (touch_temp == 0):
          $ 375 "write_port_register(138,0)"
          write_port_register(138,0)
          $ 376 "get_touch_position"
          $ 377 "get pre-positions"
          $ 378 "If read_port_register(work_type_165)≟2"
          if ( read_port_register (work_type_165) == 2):
            $ 379 "freedrive touch"
            $ 380 "move_i≔1"
            global move_i=1
            $ 381 "Loop move_i<9"
            while (move_i<9):
              $ 382 "Wait: 0.1"
              sleep(0.1)
              $ 383 "Wait save_tool=LO"
              while (get_tool_digital_in(0) == True):
                sync()
              end
              $ 384 "If A_Touch_trig_l[move_i]≟ True "
              if (A_Touch_trig_l[move_i] ==   True  ):
                $ 385 "If move_i≟A_HOR"
                if (move_i == A_HOR):
                  $ 386 "If b1_cell_info_L≟B or b1_cell_info_L≟D or b1_cell_info_L≟d or A_Prepos_l[A_VL1]≟p[0,0,0,0,0,0]"
                  if (b1_cell_info_L == B  or  b1_cell_info_L == D  or  b1_cell_info_L == d  or  A_Prepos_l[A_VL1] == p[0,0,0,0,0,0]):
                    $ 387 "write_port_register(touch_cell_155,5)"
                    write_port_register(touch_cell_155,5)
                    $ 388 "write_port_register(touch_num_156,1)"
                    write_port_register(touch_num_156,1)
                    $ 389 "Call touch_sub"
                    touch_sub()
                    $ 390 "g_cp≔get_actual_tcp_pose()"
                    global g_cp= get_actual_tcp_pose ()
                    $ 391 "If g_cp[2]<(get_margin_z+a7_cell_bottom)/1000"
                    if (g_cp[2]<(get_margin_z+a7_cell_bottom)/1000):
                      $ 392 "g_cp[2]=(get_margin_z+a7_cell_bottom)/1000"
                      g_cp[2]=(get_margin_z+a7_cell_bottom)/1000
                    end
                    $ 393 "A_Prepos_l[move_i]=g_cp"
                    A_Prepos_l[move_i]=g_cp
                  end
                else:
                  $ 394 "ElseIf move_i≟A_HOR_ML"
                  if (move_i == A_HOR_ML):
                    $ 395 "If b1_cell_info_L≟B or b1_cell_info_L≟D or b1_cell_info_L≟d or A_Prepos_l[A_VL1]≟p[0,0,0,0,0,0]"
                    if (b1_cell_info_L == B  or  b1_cell_info_L == D  or  b1_cell_info_L == d  or  A_Prepos_l[A_VL1] == p[0,0,0,0,0,0]):
                      $ 396 "write_port_register(touch_cell_155,5)"
                      write_port_register(touch_cell_155,5)
                      $ 397 "write_port_register(touch_num_156,3)"
                      write_port_register(touch_num_156,3)
                      $ 398 "Call touch_sub"
                      touch_sub()
                      $ 399 "g_cp≔get_actual_tcp_pose()"
                      global g_cp= get_actual_tcp_pose ()
                      $ 400 "If g_cp[2]<(get_margin_z+a7_cell_bottom)/1000"
                      if (g_cp[2]<(get_margin_z+a7_cell_bottom)/1000):
                        $ 401 "g_cp[2]=(get_margin_z+a7_cell_bottom)/1000"
                        g_cp[2]=(get_margin_z+a7_cell_bottom)/1000
                      end
                      $ 402 "A_Prepos_l[move_i]=g_cp"
                      A_Prepos_l[move_i]=g_cp
                    end
                  else:
                    $ 403 "ElseIf move_i≟A_HOR_R"
                    if (move_i == A_HOR_R):
                      $ 404 "If b1_cell_info_L≟B or b1_cell_info_L≟D or b1_cell_info_L≟d or A_Prepos_l[A_VL1]≟p[0,0,0,0,0,0]"
                      if (b1_cell_info_L == B  or  b1_cell_info_L == D  or  b1_cell_info_L == d  or  A_Prepos_l[A_VL1] == p[0,0,0,0,0,0]):
                        $ 405 "write_port_register(touch_cell_155,5)"
                        write_port_register(touch_cell_155,5)
                        $ 406 "write_port_register(touch_num_156,2)"
                        write_port_register(touch_num_156,2)
                        $ 407 "Call touch_sub"
                        touch_sub()
                        $ 408 "g_cp≔get_actual_tcp_pose()"
                        global g_cp= get_actual_tcp_pose ()
                        $ 409 "If g_cp[2]<(get_margin_z+a7_cell_bottom)/1000"
                        if (g_cp[2]<(get_margin_z+a7_cell_bottom)/1000):
                          $ 410 "g_cp[2]=(get_margin_z+a7_cell_bottom)/1000"
                          g_cp[2]=(get_margin_z+a7_cell_bottom)/1000
                        end
                        $ 411 "A_Prepos_l[move_i]=g_cp"
                        A_Prepos_l[move_i]=g_cp
                      end
                    else:
                      $ 412 "ElseIf move_i≟A_HOR_MR"
                      if (move_i == A_HOR_MR):
                        $ 413 "If b1_cell_info_L≟B or b1_cell_info_L≟D or b1_cell_info_L≟d or A_Prepos_l[A_VL1]≟p[0,0,0,0,0,0]"
                        if (b1_cell_info_L == B  or  b1_cell_info_L == D  or  b1_cell_info_L == d  or  A_Prepos_l[A_VL1] == p[0,0,0,0,0,0]):
                          $ 414 "write_port_register(touch_cell_155,5)"
                          write_port_register(touch_cell_155,5)
                          $ 415 "write_port_register(touch_num_156,4)"
                          write_port_register(touch_num_156,4)
                          $ 416 "Call touch_sub"
                          touch_sub()
                          $ 417 "g_cp≔get_actual_tcp_pose()"
                          global g_cp= get_actual_tcp_pose ()
                          $ 418 "If g_cp[2]<(get_margin_z+a7_cell_bottom)/1000"
                          if (g_cp[2]<(get_margin_z+a7_cell_bottom)/1000):
                            $ 419 "g_cp[2]=(get_margin_z+a7_cell_bottom)/1000"
                            g_cp[2]=(get_margin_z+a7_cell_bottom)/1000
                          end
                          $ 420 "A_Prepos_l[move_i]=g_cp"
                          A_Prepos_l[move_i]=g_cp
                        end
                      else:
                        $ 421 "Else" "noBreak"
                        $ 422 "write_port_register(touch_cell_155,move_i)"
                        write_port_register(touch_cell_155,move_i)
                        $ 423 "write_port_register(touch_num_156,1)"
                        write_port_register(touch_num_156,1)
                        $ 424 "Call touch_sub"
                        touch_sub()
                        $ 425 "A_Prepos_l[move_i]=get_actual_tcp_pose()"
                        A_Prepos_l[move_i]= get_actual_tcp_pose ()
                        $ 426 "If move_i≤4"
                        if (move_i <= 4):
                          $ 427 "write_port_register(touch_cell_155,move_i)"
                          write_port_register(touch_cell_155,move_i)
                          $ 428 "write_port_register(touch_num_156,2)"
                          write_port_register(touch_num_156,2)
                          $ 429 "Wait: 0.1"
                          sleep(0.1)
                          $ 430 "Call touch_sub"
                          touch_sub()
                          $ 431 "A_Prepos_l[move_i+9]=get_actual_tcp_pose()"
                          A_Prepos_l[move_i+9]= get_actual_tcp_pose ()
                        end
                      end
                    end
                  end
                end
              else:
                $ 432 "Else" "noBreak"
                $ 433 "A_Prepos_l[move_i]=p[0,0,0,0,0,0]"
                A_Prepos_l[move_i]=p[0,0,0,0,0,0]
                $ 434 "If move_i≤4"
                if (move_i <= 4):
                  $ 435 "A_Prepos_l[move_i+7]=p[0,0,0,0,0,0]"
                  A_Prepos_l[move_i+7]=p[0,0,0,0,0,0]
                else:
                  $ 436 "ElseIf move_i≟A_HOR"
                  if (move_i == A_HOR):
                    $ 437 "A_Prepos_l[A_HOR_ML]=p[0,0,0,0,0,0]"
                    A_Prepos_l[A_HOR_ML]=p[0,0,0,0,0,0]
                    $ 438 "A_Prepos_l[A_HOR_MR]=p[0,0,0,0,0,0]"
                    A_Prepos_l[A_HOR_MR]=p[0,0,0,0,0,0]
                    $ 439 "A_Prepos_l[A_HOR_M]=p[0,0,0,0,0,0]"
                    A_Prepos_l[A_HOR_M]=p[0,0,0,0,0,0]
                    $ 440 "A_Prepos_l[A_HOR_R]=p[0,0,0,0,0,0]"
                    A_Prepos_l[A_HOR_R]=p[0,0,0,0,0,0]
                  end
                end
              end
              $ 441 "move_i≔move_i+1"
              global move_i=move_i+1
            end
            $ 442 "change deg"
            $ 443 "move_i≔1"
            global move_i=1
            $ 444 "Loop move_i<14"
            while (move_i<14):
              $ 445 "If A_Prepos_l[move_i]≠p[0,0,0,0,0,0]"
              if (A_Prepos_l[move_i] != p[0,0,0,0,0,0]):
                $ 446 "If move_i≟A_VL1 or move_i≟A_VL2 or move_i≟A_VL1_END or move_i≟A_VL2_END"
                if (move_i == A_VL1  or  move_i == A_VL2  or  move_i == A_VL1_END  or  move_i == A_VL2_END):
                  $ 447 "b2_left_par≔ True "
                  global b2_left_par=  True
                  $ 448 "b8_wv_2f≔ False "
                  global b8_wv_2f=  False
                  $ 449 "get_pos≔A_Prepos_l[move_i]"
                  global get_pos=A_Prepos_l[move_i]
                  $ 450 "get_org≔left"
                  global get_org=p[.480496318984, .411279115151, .006998291210, -2.211681476386, -.899147924387, -1.383032568605]
                  $ 451 "get_pos≔p[get_pos[0],get_pos[1],get_pos[2],get_org[3],get_org[4],get_org[5]]"
                  global get_pos=p[get_pos[0],get_pos[1],get_pos[2],get_org[3],get_org[4],get_org[5]]
                  $ 452 "pre_tp≔tilt_3f_fun(get_pos,[0,0],a5_f_hole[1])"
                  global pre_tp=tilt_3f_fun(get_pos,[0,0],a5_f_hole[1])
                else:
                  $ 453 "ElseIf move_i≟A_VR1 or move_i≟A_VR2 or move_i≟A_VR1_END or move_i≟A_VR2_END"
                  if (move_i == A_VR1  or  move_i == A_VR2  or  move_i == A_VR1_END  or  move_i == A_VR2_END):
                    $ 454 "b2_left_par≔ False "
                    global b2_left_par=  False
                    $ 455 "b8_wv_2f≔ False "
                    global b8_wv_2f=  False
                    $ 456 "get_pos≔A_Prepos_l[move_i]"
                    global get_pos=A_Prepos_l[move_i]
                    $ 457 "get_org≔right"
                    global get_org=p[.475000000000, -.421403215678, .026417194146, 1.917761036827, -1.141682393512, 1.523356199292]
                    $ 458 "get_pos≔p[get_pos[0],get_pos[1],get_pos[2],get_org[3],get_org[4],get_org[5]]"
                    global get_pos=p[get_pos[0],get_pos[1],get_pos[2],get_org[3],get_org[4],get_org[5]]
                    $ 459 "pre_tp≔tilt_3f_fun(get_pos,[0,0],a5_f_hole[1])"
                    global pre_tp=tilt_3f_fun(get_pos,[0,0],a5_f_hole[1])
                  else:
                    $ 460 "ElseIf move_i≟A_HOR or move_i≟A_HOR_ML"
                    if (move_i == A_HOR  or  move_i == A_HOR_ML):
                      $ 461 "b8_wv_2f≔ True "
                      global b8_wv_2f=  True
                      $ 462 "b2_left_par≔ True "
                      global b2_left_par=  True
                      $ 463 "get_pos≔A_Prepos_l[move_i]"
                      global get_pos=A_Prepos_l[move_i]
                      $ 464 "get_org≔up_left"
                      global get_org=p[.492775857339, .409517380626, -.029063830209, -2.419264859926, -.998084331190, -1.368689080860]
                      $ 465 "get_pos≔p[get_pos[0],get_pos[1],get_pos[2],get_org[3],get_org[4],get_org[5]]"
                      global get_pos=p[get_pos[0],get_pos[1],get_pos[2],get_org[3],get_org[4],get_org[5]]
                      $ 466 "pre_tp≔tilt_2f_fun(get_pos,[0,0], True , True )"
                      global pre_tp=tilt_2f_fun(get_pos,[0,0],  True  ,  True  )
                    else:
                      $ 467 "ElseIf move_i≟A_HOR_R or move_i≟A_HOR_MR"
                      if (move_i == A_HOR_R  or  move_i == A_HOR_MR):
                        $ 468 "b8_wv_2f≔ True "
                        global b8_wv_2f=  True
                        $ 469 "b2_left_par≔ False "
                        global b2_left_par=  False
                        $ 470 "get_pos≔A_Prepos_l[move_i]"
                        global get_pos=A_Prepos_l[move_i]
                        $ 471 "get_org≔up_right"
                        global get_org=p[.445203173045, -.406687378356, -.031125942276, 2.308490741423, -1.066468937023, 1.322151316133]
                        $ 472 "get_pos≔p[get_pos[0],get_pos[1],get_pos[2],get_org[3],get_org[4],get_org[5]]"
                        global get_pos=p[get_pos[0],get_pos[1],get_pos[2],get_org[3],get_org[4],get_org[5]]
                        $ 473 "pre_tp≔tilt_2f_fun(get_pos,[0,0], False , True )"
                        global pre_tp=tilt_2f_fun(get_pos,[0,0],  False  ,  True  )
                      end
                    end
                  end
                end
                $ 474 "A_Prepos_l[move_i]=pre_tp"
                A_Prepos_l[move_i]=pre_tp
              end
              $ 475 "move_i≔move_i+1"
              global move_i=move_i+1
            end
            $ 476 "homeing()"
            homeing()
            $ 477 "Wait read_port_register(170)≟1"
            while (not( read_port_register (170) == 1)):
              sync()
            end
            $ 478 "write_port_register(170,0)"
            write_port_register(170,0)
          else:
            $ 479 "Else" "noBreak"
            $ 480 "value from pendant"
            $ 481 "move_i≔1"
            global move_i=1
            $ 483 "Touch_FrontandSide"
            $ 484 "If EXT_flag1[11]≟ True "
            if (EXT_flag1[11] ==   True  ):
              $ 485 "Touch front and side_Right"
              $ 486 "move_center≔pose_add(first_p_wp, p[-first_p_wp[0]+(get_center-work_touch_dis)/1000,0,0,0,0,0])"
              global move_center= pose_add (first_p_wp, p[-first_p_wp[0]+(get_center-work_touch_dis)/1000,0,0,0,0,0])
              $ 487 "get_pose_side_t≔0"
              global get_pose_side_t=0
              $ 489 "move_center[2]=(center_height+a7_cell_bottom)/1000"
              move_center[2]=(center_height+a7_cell_bottom)/1000
              $ 491 "MoveL"
              $ 492 "move_center" "breakAfter"
              movel(pose_trans(Base, move_center), a=0.5, v=0.15)
              $ 493 "touch_center≔contact_fun(p[0,0,0,0,0,0],[1,0,0],20000,20,20)"
              global touch_center=contact_fun(p[0,0,0,0,0,0],[1,0,0],20000,20,20)
              $ 494 "direction(p[0,0,0,0,0,0],[-1,0,0],10,180,200)"
              direction(p[0,0,0,0,0,0],[-1,0,0],10,180,200)
              $ 495 "get_center≔touch_center[0]*1000"
              global get_center=touch_center[0]*1000
              $ 496 "a7_f_distance≔get_center"
              global a7_f_distance=get_center
              $ 497 "move_center≔pose_add(move_center,p[0,sec_touch_dis/1000,0,0,0,0])"
              global move_center= pose_add (move_center,p[0,sec_touch_dis/1000,0,0,0,0])
              $ 498 "move_center[0]=touch_center[0]-20/1000"
              move_center[0]=touch_center[0]-20/1000
              $ 499 "MoveL"
              $ 500 "move_center" "breakAfter"
              movel(pose_trans(Base, move_center), a=0.5, v=0.15)
              $ 501 "touch_center2≔contact_fun(p[0,0,0,0,0,0],[1,0,0],20000,20,20)"
              global touch_center2=contact_fun(p[0,0,0,0,0,0],[1,0,0],20000,20,20)
              $ 502 "center_line≔get_feature_Line(touch_center,touch_center2)"
              global center_line=get_feature_Line(touch_center,touch_center2)
              $ 503 "event_cal_on≔ True "
              global event_cal_on=  True
              $ 504 "direction(p[0,0,0,0,0,0],[-1,0,0],10,180,200)"
              direction(p[0,0,0,0,0,0],[-1,0,0],10,180,200)
              $ 506 "homeing()"
              homeing()
              $ 507 "b2_left_par≔ False "
              global b2_left_par=  False
              $ 508 "b8_wv_2f≔ False "
              global b8_wv_2f=  False
              $ 509 "b2_cell≔b1_cell_info_R"
              global b2_cell=b1_cell_info_R
              $ 510 "get_pos≔get_lr(side_p_R,a6_f_width,[35,0,0,0,0],a7_f_distance,b2_left_par,b8_wv_2f,Touch_dis,get_margin_z,get_pose_side_t,30,0,center_line, True )"
              global get_pos=get_lr(p[.471584857321, -.427242166643, .026448165242, 1.806736638758, -1.227818761912, 1.383474453522],a6_f_width,[35,0,0,0,0],a7_f_distance,b2_left_par,b8_wv_2f,Touch_dis,get_margin_z,get_pose_side_t,30,0,center_line,  True  )
              $ 512 "pre_tp≔get_pos"
              global pre_tp=get_pos
              $ 513 "pre_tp≔pose_add(pre_tp, p[side_pos_x/1000,0,0,0,0,0])"
              global pre_tp= pose_add (pre_tp, p[side_pos_x/1000,0,0,0,0,0])
              $ 514 "pre_tp[2]=(center_height+a7_cell_bottom)/1000"
              pre_tp[2]=(center_height+a7_cell_bottom)/1000
              $ 515 "MoveL"
              $ 516 "pre_tp" "breakAfter"
              movel(pose_trans(Base, pre_tp), a=1.2, v=0.25)
              $ 517 "touch_side≔contact_fun(p[0,0,0,0,0,0],[0,-1,0],20000,13,13)"
              global touch_side=contact_fun(p[0,0,0,0,0,0],[0,-1,0],20000,13,13)
              $ 518 "touch_side≔get_feature_pose(touch_side,center_line)"
              global touch_side=get_feature_pose(touch_side,center_line)
              $ 519 "direction(p[0,0,0,0,0,0],[0,1,0],10,180,200)"
              direction(p[0,0,0,0,0,0],[0,1,0],10,180,200)
              $ 520 "write_welder(4, False )"
              write_welder(4,  False  )
              $ 521 "get_pose_side_t≔touch_side[1]*1000"
              global get_pose_side_t=touch_side[1]*1000
              $ 522 "get_pose_side_t≔get_pose_side_t+(a6_f_width/2)"
              global get_pose_side_t=get_pose_side_t+(a6_f_width/2)
              $ 523 "event_side_on≔ True "
              global event_side_on=  True
              $ 524 "MoveL"
              $ 525 "Direction: Base"
              global move_thread_flag_525=0
              thread move_thread_525():
                enter_critical
                move_thread_flag_525 = 1
                local towardsPos=calculate_point_to_move_towards(p[0.0,0.0,0.0,0.0,0.0,0.0], [-1,1,0], 0.03)
                movel(towardsPos, a=0.08, v=0.05)
                move_thread_flag_525 = 2
                exit_critical
              end
              move_thread_flag_525 = 0
              move_thread_han_525 = run move_thread_525()
              while (True):
                sleep(1.0E-10)
                if (move_thread_flag_525 > 1):
                  join move_thread_han_525
                  $ 526 "Until (distance)"
                  break
                end
                sync()
              end
              $ 527 "homeing()"
              homeing()
            else:
              $ 528 "Else" "noBreak"
              $ 529 "Touch front and side_Left"
              $ 530 "move_center≔pose_add(first_p_wp, p[-first_p_wp[0]+(get_center-work_touch_dis)/1000,0,0,0,0,0])"
              global move_center= pose_add (first_p_wp, p[-first_p_wp[0]+(get_center-work_touch_dis)/1000,0,0,0,0,0])
              $ 531 "get_pose_side_t≔0"
              global get_pose_side_t=0
              $ 533 "move_center[2]=(center_height+a7_cell_bottom)/1000"
              move_center[2]=(center_height+a7_cell_bottom)/1000
              $ 535 "MoveL"
              $ 536 "move_center" "breakAfter"
              movel(pose_trans(Base, move_center), a=0.5, v=0.15)
              $ 537 "touch_center≔contact_fun(p[0,0,0,0,0,0],[1,0,0],20000,20,20)"
              global touch_center=contact_fun(p[0,0,0,0,0,0],[1,0,0],20000,20,20)
              $ 538 "direction(p[0,0,0,0,0,0],[-1,0,0],10,180,200)"
              direction(p[0,0,0,0,0,0],[-1,0,0],10,180,200)
              $ 539 "get_center≔touch_center[0]*1000"
              global get_center=touch_center[0]*1000
              $ 540 "a7_f_distance≔get_center"
              global a7_f_distance=get_center
              $ 541 "move_center≔pose_add(move_center,p[0,sec_touch_dis/1000,0,0,0,0])"
              global move_center= pose_add (move_center,p[0,sec_touch_dis/1000,0,0,0,0])
              $ 542 "move_center[0]=touch_center[0]-20/1000"
              move_center[0]=touch_center[0]-20/1000
              $ 543 "MoveL"
              $ 544 "move_center" "breakAfter"
              movel(pose_trans(Base, move_center), a=0.5, v=0.15)
              $ 545 "touch_center2≔contact_fun(p[0,0,0,0,0,0],[1,0,0],20000,20,20)"
              global touch_center2=contact_fun(p[0,0,0,0,0,0],[1,0,0],20000,20,20)
              $ 546 "center_line≔get_feature_Line(touch_center,touch_center2)"
              global center_line=get_feature_Line(touch_center,touch_center2)
              $ 547 "event_cal_on≔ True "
              global event_cal_on=  True
              $ 548 "direction(p[0,0,0,0,0,0],[-1,0,0],10,180,200)"
              direction(p[0,0,0,0,0,0],[-1,0,0],10,180,200)
              $ 550 "homeing()"
              homeing()
              $ 551 "b2_left_par≔ True "
              global b2_left_par=  True
              $ 552 "b8_wv_2f≔ False "
              global b8_wv_2f=  False
              $ 553 "b2_cell≔b1_cell_info_L"
              global b2_cell=b1_cell_info_L
              $ 554 "get_pos≔get_lr(side_p_L,a6_f_width,[35,0,0,0,0],a7_f_distance,b2_left_par,b8_wv_2f,Touch_dis,get_margin_z,get_pose_side_t,30,0,center_line, True )"
              global get_pos=get_lr(p[.411215372122, .375785944375, -.010176539343, -1.953488355698, -1.125710367676, -1.228829273458],a6_f_width,[35,0,0,0,0],a7_f_distance,b2_left_par,b8_wv_2f,Touch_dis,get_margin_z,get_pose_side_t,30,0,center_line,  True  )
              $ 556 "pre_tp≔get_pos"
              global pre_tp=get_pos
              $ 557 "pre_tp≔pose_add(pre_tp, p[side_pos_x/1000,0,0,0,0,0])"
              global pre_tp= pose_add (pre_tp, p[side_pos_x/1000,0,0,0,0,0])
              $ 558 "pre_tp[2]=(center_height+a7_cell_bottom)/1000"
              pre_tp[2]=(center_height+a7_cell_bottom)/1000
              $ 559 "MoveL"
              $ 560 "pre_tp" "breakAfter"
              movel(pose_trans(Base, pre_tp), a=1.2, v=0.25)
              $ 561 "touch_side≔contact_fun(p[0,0,0,0,0,0],[0,1,0],20000,13,13)"
              global touch_side=contact_fun(p[0,0,0,0,0,0],[0,1,0],20000,13,13)
              $ 562 "touch_side≔get_feature_pose(touch_side,center_line)"
              global touch_side=get_feature_pose(touch_side,center_line)
              $ 563 "direction(p[0,0,0,0,0,0],[0,-1,0],10,180,200)"
              direction(p[0,0,0,0,0,0],[0,-1,0],10,180,200)
              $ 564 "write_welder(4, False )"
              write_welder(4,  False  )
              $ 565 "get_pose_side_t≔touch_side[1]*1000"
              global get_pose_side_t=touch_side[1]*1000
              $ 566 "get_pose_side_t≔get_pose_side_t-(a6_f_width/2)"
              global get_pose_side_t=get_pose_side_t-(a6_f_width/2)
              $ 567 "event_side_on≔ True "
              global event_side_on=  True
              $ 568 "MoveL"
              $ 569 "Direction: Base"
              global move_thread_flag_569=0
              thread move_thread_569():
                enter_critical
                move_thread_flag_569 = 1
                local towardsPos=calculate_point_to_move_towards(p[0.0,0.0,0.0,0.0,0.0,0.0], [-1,-1,0], 0.03)
                movel(towardsPos, a=0.08, v=0.05)
                move_thread_flag_569 = 2
                exit_critical
              end
              move_thread_flag_569 = 0
              move_thread_han_569 = run move_thread_569()
              while (True):
                sleep(1.0E-10)
                if (move_thread_flag_569 > 1):
                  join move_thread_han_569
                  $ 570 "Until (distance)"
                  break
                end
                sync()
              end
              $ 571 "homeing()"
              homeing()
            end
            $ 573 "Wait event_side_on≟ False "
            while (not(event_side_on ==   False  )):
              sync()
            end
          end
          $ 574 "move and touch"
          $ 575 "Touch Move"
          $ 576 "HOR_L"
          $ 577 "If A_Prepos_l[A_HOR]≠p[0,0,0,0,0,0]"
          if (A_Prepos_l[A_HOR] != p[0,0,0,0,0,0]):
            $ 578 "b2_left_par≔ True "
            global b2_left_par=  True
            $ 579 "b8_wv_2f≔ True "
            global b8_wv_2f=  True
            $ 580 "b7_tilt_degree≔[0,0,0]"
            global b7_tilt_degree=[0,0,0]
            $ 581 "A_sel_v≔A_HOR"
            global A_sel_v=A_HOR
            $ 582 "wv_direction≔1"
            global wv_direction=1
            $ 583 "Call MoveandTouchFun_2f"
            MoveandTouchFun_2f()
            $ 585 "If b1_cell_info_L≟A or b1_cell_info_L≟C or b1_cell_info_L≟c"
            if (b1_cell_info_L == A  or  b1_cell_info_L == C  or  b1_cell_info_L == c):
              $ 586 "If A_Prepos_l[A_VL1]≟p[0,0,0,0,0,0]"
              if (A_Prepos_l[A_VL1] == p[0,0,0,0,0,0]):
                $ 588 "g_tp≔A_Prepos_l[A_HOR]"
                global g_tp=A_Prepos_l[A_HOR]
                $ 591 "Folder"
                $ 592 "g_cp≔get_actual_tcp_pose()"
                global g_cp= get_actual_tcp_pose ()
                $ 593 "g_cp≔pose_trans(g_cp, p[0,0,0,d2r(12),d2r(5),0])"
                global g_cp= pose_trans (g_cp, p[0,0,0,d2r(12),d2r(5),0])
                $ 594 "MoveL"
                $ 595 "g_cp" "breakAfter"
                movel(pose_trans(Base, g_cp), a=0.08, v=0.08)
                $ 596 "for_x_HOR≔contact_fun(A_Touch_p[A_sel_v],[-1*wv_direction,0,0],10000,15,15,  False)"
                global for_x_HOR=contact_fun(A_Touch_p[A_sel_v],[-1*wv_direction,0,0],10000,15,15,  False)
                $ 597 "direction(p[0,0,0,0,0,0],[0,-1,0],20,120,160)"
                direction(p[0,0,0,0,0,0],[0,-1,0],20,120,160)
                $ 598 "write_welder(4, False )"
                write_welder(4,  False  )
              else:
                $ 599 "Else" "noBreak"
                $ 600 "for_x_HOR≔p[0,0,0,0,0,0]"
                global for_x_HOR=p[0,0,0,0,0,0]
              end
            else:
              $ 601 "ElseIf b1_cell_info_L≟E"
              if (b1_cell_info_L == E):
                $ 602 "direction(p[0,0,0,0,0,0],[0,1,0],40,120,160)"
                direction(p[0,0,0,0,0,0],[0,1,0],40,120,160)
                $ 603 "direction(p[0,0,0,0,0,0],[1,0,0],20,120,160)"
                direction(p[0,0,0,0,0,0],[1,0,0],20,120,160)
                $ 604 "for_x_HOR≔contact_fun(A_Touch_p[A_sel_v],[0,-1,0],10000,15,15,  False)"
                global for_x_HOR=contact_fun(A_Touch_p[A_sel_v],[0,-1,0],10000,15,15,  False)
                $ 605 "write_welder(4, False )"
                write_welder(4,  False  )
                $ 606 "direction(p[0,0,0,0,0,0],[0,1,0],20,120,160)"
                direction(p[0,0,0,0,0,0],[0,1,0],20,120,160)
                $ 607 "direction(p[0,0,0,0,0,0],[-1,0,0],40,120,160)"
                direction(p[0,0,0,0,0,0],[-1,0,0],40,120,160)
              end
            end
            $ 608 "If point_dist(A_Prepos_l[A_HOR], A_Prepos_l[A_VL1])>0.03"
            if (point_dist(A_Prepos_l[A_HOR], A_Prepos_l[A_VL1])>0.03):
              $ 609 "homeing()"
              homeing()
            end
          end
          $ 610 "VL1"
          $ 611 "If A_Prepos_l[A_VL1]≠p[0,0,0,0,0,0]"
          if (A_Prepos_l[A_VL1] != p[0,0,0,0,0,0]):
            $ 612 "b2_left_par≔ True "
            global b2_left_par=  True
            $ 613 "b8_wv_2f≔ False "
            global b8_wv_2f=  False
            $ 614 "b7_tilt_degree≔[0,0,0]"
            global b7_tilt_degree=[0,0,0]
            $ 615 "A_sel_v≔A_VL1"
            global A_sel_v=A_VL1
            $ 616 "A_sel_v_end≔A_VL1_END"
            global A_sel_v_end=A_VL1_END
            $ 617 "b2_par_cd≔0"
            global b2_par_cd=0
            $ 618 "If b1_cell_info_L≟A or b1_cell_info_L≟C or b1_cell_info_L≟c"
            if (b1_cell_info_L == A  or  b1_cell_info_L == C  or  b1_cell_info_L == c):
              $ 619 "Scallup_check≔ True "
              global Scallup_check=  True
            else:
              $ 620 "Else" "noBreak"
              $ 621 "Scallup_check≔ False "
              global Scallup_check=  False
            end
            $ 622 "Call MoveandTouchFun_3f"
            MoveandTouchFun_3f()
            $ 623 "If b1_cell_info_L≟A or b1_cell_info_L≟C or b1_cell_info_L≟c"
            if (b1_cell_info_L == A  or  b1_cell_info_L == C  or  b1_cell_info_L == c):
              $ 624 "If A_Prepos_l[A_HOR]≟p[0,0,0,0,0,0]"
              if (A_Prepos_l[A_HOR] == p[0,0,0,0,0,0]):
                $ 625 "direction(p[0,0,0,0,0,0],[0,-1,0],8,120,160)"
                direction(p[0,0,0,0,0,0],[0,-1,0],8,120,160)
                $ 627 "AAgcp≔get_actual_tcp_pose()"
                global AAgcp= get_actual_tcp_pose ()
                $ 628 "AAgangle≔up_left"
                global AAgangle=p[.492775857339, .409517380626, -.029063830209, -2.419264859926, -.998084331190, -1.368689080860]
                $ 629 "AAgtp≔p[AAgcp[0],AAgcp[1],AAgcp[2],AAgangle[3],AAgangle[4],AAgangle[5]]"
                global AAgtp=p[AAgcp[0],AAgcp[1],AAgcp[2],AAgangle[3],AAgangle[4],AAgangle[5]]
                $ 630 "MoveL"
                $ 631 "AAgtp" "breakAfter"
                movel(pose_trans(Base, AAgtp), a=0.08, v=0.08)
                $ 633 "for_z_VL1≔contact_fun(p[0,0,0,0,0,0],[0,0,-1],10000,15,15,  False)"
                global for_z_VL1=contact_fun(p[0,0,0,0,0,0],[0,0,-1],10000,15,15,  False)
                $ 634 "direction(p[0,0,0,0,0,0],[0,0,1],20,120,160)"
                direction(p[0,0,0,0,0,0],[0,0,1],20,120,160)
                $ 635 "write_welder(4, False )"
                write_welder(4,  False  )
              else:
                $ 636 "Else" "noBreak"
                $ 637 "for_z_VL1≔p[0,0,0,0,0,0]"
                global for_z_VL1=p[0,0,0,0,0,0]
              end
            end
          end
          $ 638 "HOR_ML"
          $ 639 "If A_Prepos_l[A_HOR_ML]≠p[0,0,0,0,0,0]"
          if (A_Prepos_l[A_HOR_ML] != p[0,0,0,0,0,0]):
            $ 640 "b2_left_par≔ True "
            global b2_left_par=  True
            $ 641 "b8_wv_2f≔ True "
            global b8_wv_2f=  True
            $ 642 "b7_tilt_degree≔[0,0,0]"
            global b7_tilt_degree=[0,0,0]
            $ 643 "A_sel_v≔A_HOR_ML"
            global A_sel_v=A_HOR_ML
            $ 644 "If b1_cell_info_L≟C or b1_cell_info_L≟D"
            if (b1_cell_info_L == C  or  b1_cell_info_L == D):
              $ 645 "wv_direction≔1"
              global wv_direction=1
              $ 646 "Call MoveFun"
              MoveFun()
              $ 647 "for_cal_xy≔contact_fun(p[0,0,0,0,0,0],[1,0,0],20000,20,20)"
              global for_cal_xy=contact_fun(p[0,0,0,0,0,0],[1,0,0],20000,20,20)
              $ 648 "direction(p[0,0,0,0,0,0],[-1,0,0],15,120,160)"
              direction(p[0,0,0,0,0,0],[-1,0,0],15,120,160)
              $ 649 "direction(p[0,0,0,0,0,0],[0,-1,0],60,120,160)"
              direction(p[0,0,0,0,0,0],[0,-1,0],60,120,160)
              $ 650 "direction(p[0,0,0,0,0,0],[1,0,0],20,120,160)"
              direction(p[0,0,0,0,0,0],[1,0,0],20,120,160)
              $ 651 "for_cal_x_wel≔contact_fun(p[0,0,0,0,0,0],[0,1,0],20000,20,20)"
              global for_cal_x_wel=contact_fun(p[0,0,0,0,0,0],[0,1,0],20000,20,20)
              $ 652 "direction(p[0,0,0,0,0,0],[0,-1,0],20,120,160)"
              direction(p[0,0,0,0,0,0],[0,-1,0],20,120,160)
              $ 653 "for_cal_zl≔contact_fun(p[0,0,0,0,0,0],[0,0,-1],20000,20,20)"
              global for_cal_zl=contact_fun(p[0,0,0,0,0,0],[0,0,-1],20000,20,20)
              $ 654 "direction(p[0,0,0,0,0,0],[0,0,1],20,120,160)"
              direction(p[0,0,0,0,0,0],[0,0,1],20,120,160)
              $ 655 "If A_Prepos_l[A_VL2]≟p[0,0,0,0,0,0]"
              if (A_Prepos_l[A_VL2] == p[0,0,0,0,0,0]):
                $ 656 "for_cal_y_wel≔contact_fun(p[0,0,0,0,0,0],[1,0,0],20000,20,20)"
                global for_cal_y_wel=contact_fun(p[0,0,0,0,0,0],[1,0,0],20000,20,20)
                $ 657 "direction(p[0,0,0,0,0,0],[-1,0,0],30,120,160)"
                direction(p[0,0,0,0,0,0],[-1,0,0],30,120,160)
              end
              $ 658 "for_cal_rot≔A_Touch_p[A_HOR]"
              global for_cal_rot=A_Touch_p[A_HOR]
              $ 659 "A_Touch_p[A_sel_v]=p[for_cal_xy[0],for_cal_xy[1],for_cal_zl[2],for_cal_rot[3],for_cal_rot[4],for_cal_rot[5]]"
              A_Touch_p[A_sel_v]=p[for_cal_xy[0],for_cal_xy[1],for_cal_zl[2],for_cal_rot[3],for_cal_rot[4],for_cal_rot[5]]
              $ 660 "A_Touch_p[A_sel_v]=pose_trans(A_Touch_p[A_sel_v], p[Touch_dis/1000,0,0,0,0,0])"
              A_Touch_p[A_sel_v]= pose_trans (A_Touch_p[A_sel_v], p[Touch_dis/1000,0,0,0,0,0])
              $ 661 "write_welder(4, False )"
              write_welder(4,  False  )
            else:
              $ 662 "Else" "noBreak"
              $ 663 "wv_direction≔1"
              global wv_direction=1
              $ 664 "for_cal_rot≔A_Touch_p[A_HOR]"
              global for_cal_rot=A_Touch_p[A_HOR]
              $ 665 "Call MoveFun_cd"
              MoveFun_cd()
              $ 666 "for_cal_y_wel≔contact_fun(p[0,0,0,0,0,0],[1,0,0],20000,20,20)"
              global for_cal_y_wel=contact_fun(p[0,0,0,0,0,0],[1,0,0],20000,20,20)
              $ 667 "for_cal_y_wel[2]=for_cal_rot[2]"
              for_cal_y_wel[2]=for_cal_rot[2]
              $ 668 "dir_x_cal≔get_feature_Line(for_cal_rot,for_cal_y_wel)"
              global dir_x_cal=get_feature_Line(for_cal_rot,for_cal_y_wel)
              $ 669 "direction(p[0,0,0,0,0,0],[-1,0,0],40,120,160)"
              direction(p[0,0,0,0,0,0],[-1,0,0],40,120,160)
              $ 670 "direction(p[0,0,0,0,0,0],[0,-1,0],70,120,160)"
              direction(p[0,0,0,0,0,0],[0,-1,0],70,120,160)
              $ 671 "for_cal_y_wel≔contact_fun(p[0,0,0,0,0,0],[1,0,0],20000,20,20)"
              global for_cal_y_wel=contact_fun(p[0,0,0,0,0,0],[1,0,0],20000,20,20)
              $ 672 "direction(p[0,0,0,0,0,0],[-1,0,0],5,120,160)"
              direction(p[0,0,0,0,0,0],[-1,0,0],5,120,160)
              $ 673 "direction(p[0,0,0,0,0,0],[0,1,0],50,120,160)"
              direction(p[0,0,0,0,0,0],[0,1,0],50,120,160)
              $ 674 "direction(p[0,0,0,0,0,0],[1,0,0],7,120,160)"
              direction(p[0,0,0,0,0,0],[1,0,0],7,120,160)
              $ 675 "for_cal_x_wel≔contact_fun(p[0,0,0,0,0,0],[0,-1,0],20000,20,20)"
              global for_cal_x_wel=contact_fun(p[0,0,0,0,0,0],[0,-1,0],20000,20,20)
              $ 676 "get_ml≔get_feature_pose(for_cal_x_wel,for_cal_rot)"
              global get_ml=get_feature_pose(for_cal_x_wel,for_cal_rot)
              $ 678 "A_Touch_p[A_sel_v]=feature_offset(for_cal_rot,p[0,get_ml[0]+(-cd_offset+cd_extra_dis)/1000,0,0,0,0],dir_x_cal)"
              A_Touch_p[A_sel_v]=feature_offset(for_cal_rot,p[0,get_ml[0]+(-cd_offset+cd_extra_dis)/1000,0,0,0,0],dir_x_cal)
              $ 679 "direction(p[0,0,0,0,0,0],[0,1,0],5,120,160)"
              direction(p[0,0,0,0,0,0],[0,1,0],5,120,160)
              $ 680 "direction(p[0,0,0,0,0,0],[-1,0,0],20,120,160)"
              direction(p[0,0,0,0,0,0],[-1,0,0],20,120,160)
              $ 681 "write_welder(4, False )"
              write_welder(4,  False  )
            end
          else:
            $ 682 "Else" "noBreak"
            $ 683 "homeing()"
            homeing()
          end
          $ 684 "VL2"
          $ 685 "If A_Prepos_l[A_VL2]≠p[0,0,0,0,0,0]"
          if (A_Prepos_l[A_VL2] != p[0,0,0,0,0,0]):
            $ 686 "b2_left_par≔ True "
            global b2_left_par=  True
            $ 687 "b8_wv_2f≔ False "
            global b8_wv_2f=  False
            $ 688 "b7_tilt_degree≔basic_tilt_3f"
            global b7_tilt_degree=basic_tilt_3f
            $ 689 "A_sel_v≔A_VL2"
            global A_sel_v=A_VL2
            $ 690 "A_sel_v_end≔A_VL2_END"
            global A_sel_v_end=A_VL2_END
            $ 691 "b2_par_cd≔1"
            global b2_par_cd=1
            $ 692 "If b1_cell_info_L≟A or b1_cell_info_L≟C or b1_cell_info_L≟c"
            if (b1_cell_info_L == A  or  b1_cell_info_L == C  or  b1_cell_info_L == c):
              $ 693 "Scallup_check≔ True "
              global Scallup_check=  True
            else:
              $ 694 "Else" "noBreak"
              $ 695 "Scallup_check≔ False "
              global Scallup_check=  False
            end
            $ 696 "If b1_cell_info_L≟d or b1_cell_info_L≟c"
            if (b1_cell_info_L == d  or  b1_cell_info_L == c):
              $ 697 "Halt"
              halt
            else:
              $ 698 "Else" "noBreak"
              $ 699 "If A_Touch_p[A_VL1]≟p[0,0,0,0,0,0]"
              if (A_Touch_p[A_VL1] == p[0,0,0,0,0,0]):
                $ 700 "Call MoveandTouchFun_3f"
                MoveandTouchFun_3f()
                $ 701 "If A_Prepos_l[A_HOR_ML]≟p[0,0,0,0,0,0]"
                if (A_Prepos_l[A_HOR_ML] == p[0,0,0,0,0,0]):
                  $ 702 "direction(p[0,0,0,0,0,0],[0,-1,0],8,120,160)"
                  direction(p[0,0,0,0,0,0],[0,-1,0],8,120,160)
                  $ 703 "AAgcp≔get_actual_tcp_pose()"
                  global AAgcp= get_actual_tcp_pose ()
                  $ 704 "AAgangle≔up_left"
                  global AAgangle=p[.492775857339, .409517380626, -.029063830209, -2.419264859926, -.998084331190, -1.368689080860]
                  $ 705 "AAgtp≔p[AAgcp[0],AAgcp[1],AAgcp[2],AAgangle[3],AAgangle[4],AAgangle[5]]"
                  global AAgtp=p[AAgcp[0],AAgcp[1],AAgcp[2],AAgangle[3],AAgangle[4],AAgangle[5]]
                  $ 706 "MoveL"
                  $ 707 "AAgtp" "breakAfter"
                  movel(pose_trans(Base, AAgtp), a=0.08, v=0.08)
                  $ 709 "If b1_cell_info_L≠E and b1_cell_info_L≠e"
                  if (b1_cell_info_L != E  and  b1_cell_info_L != e):
                    $ 710 "for_cal_zl≔contact_fun(p[0,0,0,0,0,0],[0,0,-1],20000,20,20)"
                    global for_cal_zl=contact_fun(p[0,0,0,0,0,0],[0,0,-1],20000,20,20)
                    $ 711 "direction(p[0,0,0,0,0,0],[0,0,1],10,120,160)"
                    direction(p[0,0,0,0,0,0],[0,0,1],10,120,160)
                  end
                end
                $ 712 "touch_tmp≔A_Touch_p[A_sel_v]"
                global touch_tmp=A_Touch_p[A_sel_v]
                $ 713 "If b1_cell_info_L≠E and b1_cell_info_L≠e"
                if (b1_cell_info_L != E  and  b1_cell_info_L != e):
                  $ 714 "touch_tmp[2]=for_cal_zl[2]"
                  touch_tmp[2]=for_cal_zl[2]
                  $ 715 "A_Touch_p[A_sel_v]=touch_tmp"
                  A_Touch_p[A_sel_v]=touch_tmp
                end
                $ 716 "for_cal_y_wel≔A_Touch_p[A_sel_v]"
                global for_cal_y_wel=A_Touch_p[A_sel_v]
                $ 717 "for_cal_x_wel≔A_Touch_p[A_sel_v]"
                global for_cal_x_wel=A_Touch_p[A_sel_v]
              else:
                $ 718 "Else" "noBreak"
                $ 719 "Call MoveFun"
                MoveFun()
                $ 720 "for_cal_y_wel≔contact_fun(p[0,0,0,0,0,0],[1,0,0],20000,20,20)"
                global for_cal_y_wel=contact_fun(p[0,0,0,0,0,0],[1,0,0],20000,20,20)
                $ 721 "direction(p[0,0,0,0,0,0],[-1,0,0],40,120,160)"
                direction(p[0,0,0,0,0,0],[-1,0,0],40,120,160)
                $ 722 "If A_Prepos_l[A_HOR_ML]≟p[0,0,0,0,0,0]"
                if (A_Prepos_l[A_HOR_ML] == p[0,0,0,0,0,0]):
                  $ 723 "direction(p[0,0,0,0,0,0],[0,1,0],60,120,160)"
                  direction(p[0,0,0,0,0,0],[0,1,0],60,120,160)
                  $ 724 "var_2≔contact_fun(p[0,0,0,0,0,0],[1,0,0],20000,20,20)"
                  global var_2=contact_fun(p[0,0,0,0,0,0],[1,0,0],20000,20,20)
                  $ 725 "direction(p[0,0,0,0,0,0],[-1,0,0],5,120,160)"
                  direction(p[0,0,0,0,0,0],[-1,0,0],5,120,160)
                  $ 726 "direction(p[0,0,0,0,0,0],[0,-1,0],60,120,160)"
                  direction(p[0,0,0,0,0,0],[0,-1,0],60,120,160)
                  $ 727 "direction(p[0,0,0,0,0,0],[1,0,0],10,120,160)"
                  direction(p[0,0,0,0,0,0],[1,0,0],10,120,160)
                  $ 728 "for_cal_x_wel≔contact_fun(p[0,0,0,0,0,0],[0,1,0],20000,20,20)"
                  global for_cal_x_wel=contact_fun(p[0,0,0,0,0,0],[0,1,0],20000,20,20)
                  $ 729 "direction(p[0,0,0,0,0,0],[0,-1,0],20,120,160)"
                  direction(p[0,0,0,0,0,0],[0,-1,0],20,120,160)
                  $ 730 "AAgcp≔get_actual_tcp_pose()"
                  global AAgcp= get_actual_tcp_pose ()
                  $ 731 "AAgangle≔up_left"
                  global AAgangle=p[.492775857339, .409517380626, -.029063830209, -2.419264859926, -.998084331190, -1.368689080860]
                  $ 732 "AAgtp≔p[AAgcp[0],AAgcp[1],AAgcp[2],AAgangle[3],AAgangle[4],AAgangle[5]]"
                  global AAgtp=p[AAgcp[0],AAgcp[1],AAgcp[2],AAgangle[3],AAgangle[4],AAgangle[5]]
                  $ 733 "MoveL"
                  $ 734 "AAgtp" "breakAfter"
                  movel(pose_trans(Base, AAgtp), a=0.08, v=0.08)
                  $ 736 "If b1_cell_info_L≠E and b1_cell_info_L≠e"
                  if (b1_cell_info_L != E  and  b1_cell_info_L != e):
                    $ 737 "for_cal_zl≔contact_fun(p[0,0,0,0,0,0],[0,0,-1],20000,20,20)"
                    global for_cal_zl=contact_fun(p[0,0,0,0,0,0],[0,0,-1],20000,20,20)
                    $ 738 "direction(p[0,0,0,0,0,0],[0,0,1],10,120,160)"
                    direction(p[0,0,0,0,0,0],[0,0,1],10,120,160)
                  end
                  $ 739 "direction(p[0,0,0,0,0,0],[-1,0,0],20,120,160)"
                  direction(p[0,0,0,0,0,0],[-1,0,0],20,120,160)
                end
                $ 740 "for_cal_rot≔A_Touch_p[A_VL1]"
                global for_cal_rot=A_Touch_p[A_VL1]
                $ 741 "If b1_cell_info_L≠E and b1_cell_info_L≠e"
                if (b1_cell_info_L != E  and  b1_cell_info_L != e):
                  $ 742 "A_Touch_p[A_sel_v]=p[for_cal_y_wel[0],for_cal_x_wel[1],for_cal_zl[2],for_cal_rot[3],for_cal_rot[4],for_cal_rot[5]]"
                  A_Touch_p[A_sel_v]=p[for_cal_y_wel[0],for_cal_x_wel[1],for_cal_zl[2],for_cal_rot[3],for_cal_rot[4],for_cal_rot[5]]
                  $ 743 "touch_tmp=p[for_cal_y_wel[0],for_cal_x_wel[1],for_cal_zl[2],for_cal_rot[3],for_cal_rot[4],for_cal_rot[5]]"
                  touch_tmp=p[for_cal_y_wel[0],for_cal_x_wel[1],for_cal_zl[2],for_cal_rot[3],for_cal_rot[4],for_cal_rot[5]]
                else:
                  $ 744 "Else" "noBreak"
                  $ 745 "touch_tmp=p[for_cal_y_wel[0],for_cal_x_wel[1],for_cal_x_wel[2],for_cal_rot[3],for_cal_rot[4],for_cal_rot[5]]"
                  touch_tmp=p[for_cal_y_wel[0],for_cal_x_wel[1],for_cal_x_wel[2],for_cal_rot[3],for_cal_rot[4],for_cal_rot[5]]
                end
                $ 746 "If Scallup_check≟ False "
                if (Scallup_check ==   False  ):
                  $ 747 "touch_tmp≔pose_trans(touch_tmp,p[-(Touch_dis)/1000,0,0,0,0,0])"
                  global touch_tmp= pose_trans (touch_tmp,p[-(Touch_dis)/1000,0,0,0,0,0])
                  $ 748 "A_Touch_p[A_sel_v]=touch_tmp"
                  A_Touch_p[A_sel_v]=touch_tmp
                else:
                  $ 749 "Else" "noBreak"
                  $ 750 "Scallup_check≔ False "
                  global Scallup_check=  False
                end
                $ 751 "write_welder(4, False )"
                write_welder(4,  False  )
              end
            end
            $ 752 "b2_par_cd≔0"
            global b2_par_cd=0
            $ 753 "homeing()"
            homeing()
          else:
            $ 754 "Else" "noBreak"
            $ 755 "homeing()"
            homeing()
          end
          $ 756 "HOR_R"
          $ 757 "If A_Prepos_l[A_HOR_R]≠p[0,0,0,0,0,0]"
          if (A_Prepos_l[A_HOR_R] != p[0,0,0,0,0,0]):
            $ 758 "b2_left_par≔ False "
            global b2_left_par=  False
            $ 759 "b8_wv_2f≔ True "
            global b8_wv_2f=  True
            $ 760 "b7_tilt_degree≔[0,0,0]"
            global b7_tilt_degree=[0,0,0]
            $ 761 "A_sel_v≔A_HOR_R"
            global A_sel_v=A_HOR_R
            $ 762 "wv_direction≔-1"
            global wv_direction=-1
            $ 763 "Call MoveandTouchFun_2f"
            MoveandTouchFun_2f()
            $ 765 "If b1_cell_info_R≟A or b1_cell_info_R≟C or b1_cell_info_R≟c"
            if (b1_cell_info_R == A  or  b1_cell_info_R == C  or  b1_cell_info_R == c):
              $ 766 "If A_Prepos_l[A_VR1]≟p[0,0,0,0,0,0]"
              if (A_Prepos_l[A_VR1] == p[0,0,0,0,0,0]):
                $ 768 "g_tp≔A_Prepos_l[A_HOR_R]"
                global g_tp=A_Prepos_l[A_HOR_R]
                $ 769 "Folder"
                $ 770 "g_cp≔get_actual_tcp_pose()"
                global g_cp= get_actual_tcp_pose ()
                $ 771 "g_cp≔pose_trans(g_cp, p[0,0,0,d2r(-12),d2r(5),0])"
                global g_cp= pose_trans (g_cp, p[0,0,0,d2r(-12),d2r(5),0])
                $ 772 "MoveL"
                $ 773 "g_cp" "breakAfter"
                movel(pose_trans(Base, g_cp), a=0.08, v=0.08)
                $ 776 "for_x_HOR_R≔contact_fun(A_Touch_p[A_HOR_R],[-1*wv_direction,0,0],10000,15,15,  False)"
                global for_x_HOR_R=contact_fun(A_Touch_p[A_HOR_R],[-1*wv_direction,0,0],10000,15,15,  False)
                $ 777 "direction(p[0,0,0,0,0,0],[0,1,0],20,120,160)"
                direction(p[0,0,0,0,0,0],[0,1,0],20,120,160)
                $ 778 "write_welder(4, False )"
                write_welder(4,  False  )
              else:
                $ 779 "Else" "noBreak"
                $ 780 "for_x_HOR_R≔p[0,0,0,0,0,0]"
                global for_x_HOR_R=p[0,0,0,0,0,0]
              end
            end
            $ 781 "wv_direction≔1"
            global wv_direction=1
            $ 782 "If point_dist(A_Prepos_l[A_HOR_R], A_Prepos_l[A_VR1])>0.03"
            if (point_dist(A_Prepos_l[A_HOR_R], A_Prepos_l[A_VR1])>0.03):
              $ 783 "homeing()"
              homeing()
            end
          end
          $ 784 "VR1"
          $ 785 "If A_Prepos_l[A_VR1]≠p[0,0,0,0,0,0]"
          if (A_Prepos_l[A_VR1] != p[0,0,0,0,0,0]):
            $ 786 "b2_left_par≔ False "
            global b2_left_par=  False
            $ 787 "b8_wv_2f≔ False "
            global b8_wv_2f=  False
            $ 788 "b7_tilt_degree≔basic_tilt_3f"
            global b7_tilt_degree=basic_tilt_3f
            $ 789 "A_sel_v≔A_VR1"
            global A_sel_v=A_VR1
            $ 790 "A_sel_v_end≔A_VR1_END"
            global A_sel_v_end=A_VR1_END
            $ 791 "b2_par_cd≔0"
            global b2_par_cd=0
            $ 792 "If b1_cell_info_R≟A or b1_cell_info_R≟C or b1_cell_info_R≟c"
            if (b1_cell_info_R == A  or  b1_cell_info_R == C  or  b1_cell_info_R == c):
              $ 793 "Scallup_check≔ True "
              global Scallup_check=  True
            else:
              $ 794 "Else" "noBreak"
              $ 795 "Scallup_check≔ False "
              global Scallup_check=  False
            end
            $ 796 "Call MoveandTouchFun_3f"
            MoveandTouchFun_3f()
            $ 797 "If b1_cell_info_R≟A or b1_cell_info_R≟C or b1_cell_info_R≟c"
            if (b1_cell_info_R == A  or  b1_cell_info_R == C  or  b1_cell_info_R == c):
              $ 798 "If A_Prepos_l[A_HOR_R]≟p[0,0,0,0,0,0]"
              if (A_Prepos_l[A_HOR_R] == p[0,0,0,0,0,0]):
                $ 799 "direction(p[0,0,0,0,0,0],[0,1,0],8,120,160)"
                direction(p[0,0,0,0,0,0],[0,1,0],8,120,160)
                $ 800 "AAgcp≔get_actual_tcp_pose()"
                global AAgcp= get_actual_tcp_pose ()
                $ 801 "AAgangle≔up_right"
                global AAgangle=p[.445203173045, -.406687378356, -.031125942276, 2.308490741423, -1.066468937023, 1.322151316133]
                $ 802 "AAgtp≔p[AAgcp[0],AAgcp[1],AAgcp[2],AAgangle[3],AAgangle[4],AAgangle[5]]"
                global AAgtp=p[AAgcp[0],AAgcp[1],AAgcp[2],AAgangle[3],AAgangle[4],AAgangle[5]]
                $ 803 "MoveL"
                $ 804 "AAgtp" "breakAfter"
                movel(pose_trans(Base, AAgtp), a=0.08, v=0.08)
                $ 806 "for_z_VR1≔contact_fun(p[0,0,0,0,0,0],[0,0,-1],10000,15,15,  False)"
                global for_z_VR1=contact_fun(p[0,0,0,0,0,0],[0,0,-1],10000,15,15,  False)
                $ 807 "direction(p[0,0,0,0,0,0],[0,0,1],20,120,160)"
                direction(p[0,0,0,0,0,0],[0,0,1],20,120,160)
                $ 808 "write_welder(4, False )"
                write_welder(4,  False  )
              else:
                $ 809 "Else" "noBreak"
                $ 810 "for_z_VR1≔p[0,0,0,0,0,0]"
                global for_z_VR1=p[0,0,0,0,0,0]
              end
            end
          end
          $ 811 "HOR_MR"
          $ 812 "If A_Prepos_l[A_HOR_MR]≠p[0,0,0,0,0,0]"
          if (A_Prepos_l[A_HOR_MR] != p[0,0,0,0,0,0]):
            $ 813 "INIT"
            $ 814 "b2_left_par≔ False "
            global b2_left_par=  False
            $ 815 "b8_wv_2f≔ True "
            global b8_wv_2f=  True
            $ 816 "b7_tilt_degree≔[0,0,0]"
            global b7_tilt_degree=[0,0,0]
            $ 817 "A_sel_v≔A_HOR_MR"
            global A_sel_v=A_HOR_MR
            $ 818 "If b1_cell_info_R≟C or b1_cell_info_R≟D"
            if (b1_cell_info_R == C  or  b1_cell_info_R == D):
              $ 819 "wv_direction≔-1"
              global wv_direction=-1
              $ 820 "Call MoveFun_cd"
              MoveFun_cd()
              $ 821 "for_cal_xy≔contact_fun(p[0,0,0,0,0,0],[1,0,0],20000,20,20)"
              global for_cal_xy=contact_fun(p[0,0,0,0,0,0],[1,0,0],20000,20,20)
              $ 822 "direction(p[0,0,0,0,0,0],[-1,0,0],15,120,160)"
              direction(p[0,0,0,0,0,0],[-1,0,0],15,120,160)
              $ 823 "direction(p[0,0,0,0,0,0],[0,1,0],60,120,160)"
              direction(p[0,0,0,0,0,0],[0,1,0],60,120,160)
              $ 824 "direction(p[0,0,0,0,0,0],[1,0,0],20,120,160)"
              direction(p[0,0,0,0,0,0],[1,0,0],20,120,160)
              $ 825 "for_cal_x_wel≔contact_fun(p[0,0,0,0,0,0],[0,-1,0],20000,20,20)"
              global for_cal_x_wel=contact_fun(p[0,0,0,0,0,0],[0,-1,0],20000,20,20)
              $ 826 "direction(p[0,0,0,0,0,0],[0,1,0],20,120,160)"
              direction(p[0,0,0,0,0,0],[0,1,0],20,120,160)
              $ 827 "for_cal_zr≔contact_fun(p[0,0,0,0,0,0],[0,0,-1],20000,20,20)"
              global for_cal_zr=contact_fun(p[0,0,0,0,0,0],[0,0,-1],20000,20,20)
              $ 828 "direction(p[0,0,0,0,0,0],[0,0,1],20,120,160)"
              direction(p[0,0,0,0,0,0],[0,0,1],20,120,160)
              $ 829 "If A_Prepos_l[A_VR2]≟p[0,0,0,0,0,0]"
              if (A_Prepos_l[A_VR2] == p[0,0,0,0,0,0]):
                $ 830 "for_cal_y_wel≔contact_fun(p[0,0,0,0,0,0],[1,0,0],20000,20,20)"
                global for_cal_y_wel=contact_fun(p[0,0,0,0,0,0],[1,0,0],20000,20,20)
                $ 831 "direction(p[0,0,0,0,0,0],[-1,0,0],8,120,160)"
                direction(p[0,0,0,0,0,0],[-1,0,0],8,120,160)
              end
              $ 832 "for_cal_rot≔A_Touch_p[A_HOR_R]"
              global for_cal_rot=A_Touch_p[A_HOR_R]
              $ 833 "A_Touch_p[A_sel_v]=p[for_cal_xy[0],for_cal_xy[1],for_cal_zr[2],for_cal_rot[3],for_cal_rot[4],for_cal_rot[5]]"
              A_Touch_p[A_sel_v]=p[for_cal_xy[0],for_cal_xy[1],for_cal_zr[2],for_cal_rot[3],for_cal_rot[4],for_cal_rot[5]]
              $ 834 "A_Touch_p[A_sel_v]=pose_trans(A_Touch_p[A_sel_v], p[-Touch_dis/1000,0,0,0,0,0])"
              A_Touch_p[A_sel_v]= pose_trans (A_Touch_p[A_sel_v], p[-Touch_dis/1000,0,0,0,0,0])
              $ 835 "write_welder(4, False )"
              write_welder(4,  False  )
            else:
              $ 836 "Else" "noBreak"
              $ 837 "wv_direction≔-1"
              global wv_direction=-1
              $ 838 "for_cal_rot≔A_Touch_p[A_HOR_R]"
              global for_cal_rot=A_Touch_p[A_HOR_R]
              $ 839 "Call MoveFun_cd"
              MoveFun_cd()
              $ 840 "for_cal_y_wel≔contact_fun(p[0,0,0,0,0,0],[1,0,0],20000,20,20)"
              global for_cal_y_wel=contact_fun(p[0,0,0,0,0,0],[1,0,0],20000,20,20)
              $ 841 "vr2_p1≔for_cal_y_wel"
              global vr2_p1=for_cal_y_wel
              $ 842 "for_cal_y_wel[2]=for_cal_rot[2]"
              for_cal_y_wel[2]=for_cal_rot[2]
              $ 843 "dir_x_cal≔get_feature_Line(for_cal_rot,for_cal_y_wel)"
              global dir_x_cal=get_feature_Line(for_cal_rot,for_cal_y_wel)
              $ 844 "vr2_p2≔feature_offset(vr2_p1,p[0,0.02,0,0,0,0],dir_x_cal)"
              global vr2_p2=feature_offset(vr2_p1,p[0,0.02,0,0,0,0],dir_x_cal)
              $ 845 "direction(p[0,0,0,0,0,0],[-1,0,0],40,120,160)"
              direction(p[0,0,0,0,0,0],[-1,0,0],40,120,160)
              $ 846 "direction(p[0,0,0,0,0,0],[0,1,0],70,120,160)"
              direction(p[0,0,0,0,0,0],[0,1,0],70,120,160)
              $ 847 "for_cal_y_wel≔contact_fun(p[0,0,0,0,0,0],[1,0,0],20000,20,20)"
              global for_cal_y_wel=contact_fun(p[0,0,0,0,0,0],[1,0,0],20000,20,20)
              $ 848 "direction(p[0,0,0,0,0,0],[-1,0,0],5,120,160)"
              direction(p[0,0,0,0,0,0],[-1,0,0],5,120,160)
              $ 849 "direction(p[0,0,0,0,0,0],[0,-1,0],50,120,160)"
              direction(p[0,0,0,0,0,0],[0,-1,0],50,120,160)
              $ 850 "direction(p[0,0,0,0,0,0],[1,0,0],7,120,160)"
              direction(p[0,0,0,0,0,0],[1,0,0],7,120,160)
              $ 851 "for_cal_x_wel≔contact_fun(p[0,0,0,0,0,0],[0,1,0],20000,20,20)"
              global for_cal_x_wel=contact_fun(p[0,0,0,0,0,0],[0,1,0],20000,20,20)
              $ 852 "vr2_p3≔for_cal_x_wel"
              global vr2_p3=for_cal_x_wel
              $ 853 "get_ml≔get_feature_pose(for_cal_x_wel,for_cal_rot)"
              global get_ml=get_feature_pose(for_cal_x_wel,for_cal_rot)
              $ 855 "A_Touch_p[A_sel_v]=feature_offset(for_cal_rot,p[0,-get_ml[0]+(-cd_offset+cd_extra_dis)/1000,0,0,0,0],dir_x_cal)"
              A_Touch_p[A_sel_v]=feature_offset(for_cal_rot,p[0,-get_ml[0]+(-cd_offset+cd_extra_dis)/1000,0,0,0,0],dir_x_cal)
              $ 856 "vr2_p4≔A_Touch_p[A_HOR_MR]"
              global vr2_p4=A_Touch_p[A_HOR_MR]
              $ 857 "direction(p[0,0,0,0,0,0],[0,-1,0],5,120,160)"
              direction(p[0,0,0,0,0,0],[0,-1,0],5,120,160)
              $ 858 "direction(p[0,0,0,0,0,0],[-1,0,0],20,120,160)"
              direction(p[0,0,0,0,0,0],[-1,0,0],20,120,160)
              $ 859 "write_welder(4, False )"
              write_welder(4,  False  )
            end
            $ 860 "wv_direction≔1"
            global wv_direction=1
          end
          $ 861 "VR2"
          $ 862 "If A_Prepos_l[A_VR2]≠p[0,0,0,0,0,0]"
          if (A_Prepos_l[A_VR2] != p[0,0,0,0,0,0]):
            $ 863 "Init"
            $ 864 "b2_left_par≔ False "
            global b2_left_par=  False
            $ 865 "b8_wv_2f≔ False "
            global b8_wv_2f=  False
            $ 866 "b7_tilt_degree≔basic_tilt_3f"
            global b7_tilt_degree=basic_tilt_3f
            $ 867 "A_sel_v≔A_VR2"
            global A_sel_v=A_VR2
            $ 868 "A_sel_v_end≔A_VR2_END"
            global A_sel_v_end=A_VR2_END
            $ 869 "b2_par_cd≔1"
            global b2_par_cd=1
            $ 870 "If b1_cell_info_R≟A or b1_cell_info_R≟C or b1_cell_info_R≟c"
            if (b1_cell_info_R == A  or  b1_cell_info_R == C  or  b1_cell_info_R == c):
              $ 871 "Scallup_check≔ True "
              global Scallup_check=  True
            else:
              $ 872 "Else" "noBreak"
              $ 873 "Scallup_check≔ False "
              global Scallup_check=  False
            end
            $ 874 "If b1_cell_info_R≟d or b1_cell_info_R≟c"
            if (b1_cell_info_R == d  or  b1_cell_info_R == c):
              $ 875 "If vr2_p1≟p[0,0,0,0,0,0]"
              if (vr2_p1 == p[0,0,0,0,0,0]):
                $ 876 "Call MoveFun_cd"
                MoveFun_cd()
                $ 877 "vr2_p1≔contact_fun(p[0,0,0,0,0,0],[1,0,0],20000,20,20)"
                global vr2_p1=contact_fun(p[0,0,0,0,0,0],[1,0,0],20000,20,20)
                $ 878 "direction(p[0,0,0,0,0,0],[-1,0,0],20,120,160)"
                direction(p[0,0,0,0,0,0],[-1,0,0],20,120,160)
                $ 879 "direction(p[0,0,0,0,0,0],[0,1,0],10,120,160)"
                direction(p[0,0,0,0,0,0],[0,1,0],10,120,160)
                $ 880 "vr2_p2≔contact_fun(p[0,0,0,0,0,0],[1,0,0],20000,20,20)"
                global vr2_p2=contact_fun(p[0,0,0,0,0,0],[1,0,0],20000,20,20)
                $ 881 "direction(p[0,0,0,0,0,0],[-1,0,0],14,120,160)"
                direction(p[0,0,0,0,0,0],[-1,0,0],14,120,160)
                $ 882 "vr2_p3≔contact_fun(p[0,0,0,0,0,0],[0,1,0],20000,20,20)"
                global vr2_p3=contact_fun(p[0,0,0,0,0,0],[0,1,0],20000,20,20)
                $ 883 "direction(p[0,0,0,0,0,0],[0,-1,0],30,120,160)"
                direction(p[0,0,0,0,0,0],[0,-1,0],30,120,160)
                $ 884 "direction(p[0,0,0,0,0,0],[-1,0,0],20,120,160)"
                direction(p[0,0,0,0,0,0],[-1,0,0],20,120,160)
                $ 885 "vr2_p4≔contact_fun(p[0,0,0,0,0,0],[0,0,-1],20000,20,20)"
                global vr2_p4=contact_fun(p[0,0,0,0,0,0],[0,0,-1],20000,20,20)
                $ 886 "direction(p[0,0,0,0,0,0],[0,0,1],40,120,160)"
                direction(p[0,0,0,0,0,0],[0,0,1],40,120,160)
